CASE iStopStandby OF
0:
	StandbyStopR(CLK:=stopStandby);
	IF StandbyStopR.Q THEN
		iStopStandby := 5;
	END_IF
5:
	IF FSMode THEN
		FSStopStandby(IN:=TRUE,PT:=FSTime);
		IF FSStopStandby.Q THEN
			iStopStandby := 10;
			FSStopStandby(IN:=FALSE,PT:=FSTime);
		END_IF
	ELSE
		iStopStandby:=10;
	END_IF
10:
	standbyCommand := FALSE;
	stopStandbyTimer(IN:=TRUE, PT:=timeout);
		IF stopStandbyTimer.Q THEN
			stopStandbyTimer(IN:=FALSE);
			IF NOT standbyClose THEN
				IF standbyStart THEN
					criticalStandbyStopFailed := TRUE;
				END_IF
					warningStandbyNotClose := TRUE;
			END_IF
			iStopStandby := 0;
		END_IF
END_CASE


(*-------------------------------------------------------------------------------------------------------------------------------------------*)

CASE iStopThird OF
0:
	ThirdStopR(CLK:=stopThird);
	IF ThirdStopR.Q THEN
		iStopThird := 10;
	END_IF
10:
	thirdCommand := FALSE;
	stopThirdTimer(IN:=TRUE, PT:=timeout);
		IF stopThirdTimer.Q THEN
			stopThirdTimer(IN:=FALSE);
			IF NOT thirdClose THEN
				IF thirdStart THEN
					criticalThirdStopFailed := TRUE;
				END_IF
				warningThirdNotClose := TRUE;
			END_IF
			iStopThird := 0;
		END_IF
END_CASE


(*-------------------------------------------------------------------------------------------------------------------------------------------*)

SOnceDuty(CLK:=(iStopDuty = 10));
IF SOnceDuty.Q THEN
		A1^:=FALSE;
		A2^:=FALSE;
		A3^:=FALSE;
END_IF


SOnceStandby(CLK:=(iStopStandby = 10));
IF SOnceStandby.Q THEN
		B1^:=FALSE;
		B2^:=FALSE;
		B3^:=FALSE;
END_IF

IF thirdDevice THEN
SOnceThird(CLK:=(iStopThird = 10));
IF SOnceThird.Q THEN
		C1^:=FALSE;
		C2^:=FALSE;
		C3^:=FALSE;
END_IF
END_IF


(*-------------------------------------------------------------------------------------------------------------------------------------------*)

(*
IF FSMode THEN

FSBothStop(IN:=NOT dutyCommand AND NOT standbyCommand,PT:=FSBothTime);
SOnceFS(CLK:=FSBothStop.Q);
IF SOnceFS.Q THEN
	FSBothStop(IN:=FALSE,PT:=FSBothTime);
	Q1^ := TRUE;
	Q2^ := TRUE;
	Q3^:=TRUE;
END_IF

END_IF
*)
END_ACTION
ACTION test:
dutyStart := dutyCommand;
standbyStart := standbyCommand;
thirdStart:=thirdCommand;
END_ACTION

(* POU module/INLET_SCREENING_OPERATION_2_old, CFC *)
PROGRAM INLET_SCREENING_OPERATION_2_old
VAR
	bTest: BOOL;
	bTestReault: BOOL;

	LSH105B : inBlock;
	LSHH105B: inBlock;
	bPenstockDual: BOOL;
	Timer1: TON;
	bWarningStreamLineOverflow: BOOL;
	bFineScreen: BOOL;
	F101B: fb_equipment_with_linking;
	XV101B1 : fb_equipment_with_linking;
	StopTimer: TON;
	bScrewConveyor: BOOL;
	bScreenCompactor: BOOL;
	bWaterSprayScreenDuty: BOOL;
	bWaterSprayScreenStandby: BOOL;
	bPenstockDuty: BOOL;
	bPenstockStandby: BOOL;
	XV101B2: fb_equipment_with_linking;
	timerCompactor: TON;
	bFineScreenDual: BOOL;
	PS101B: fb_equipment_with_linking;
	bContinuousWaterSpray: BOOL;
	C102B: fb_equipment_with_linking;
	C101B: fb_equipment_with_linking;
	XV102B: fb_equipment_with_linking;
END_VAR
VAR (* helpers for the ST form of the networks *)
	_en57 : BOOL;
	_t57 : BOOL;
	_en85 : BOOL;
	_t85 : BOOL;
END_VAR
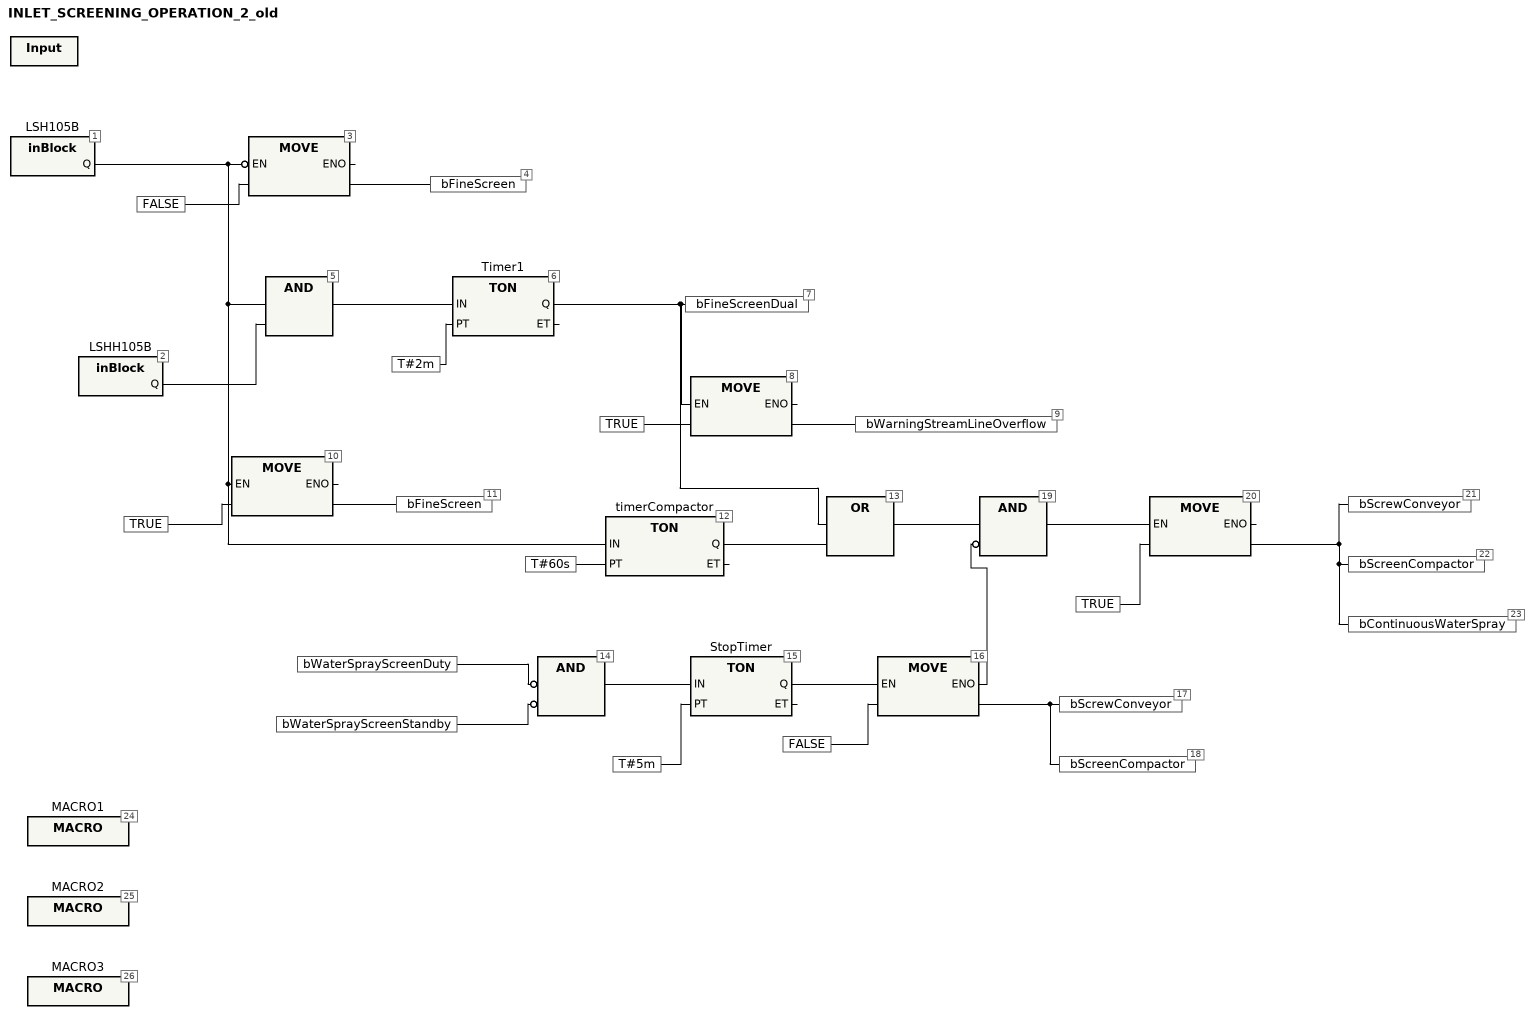
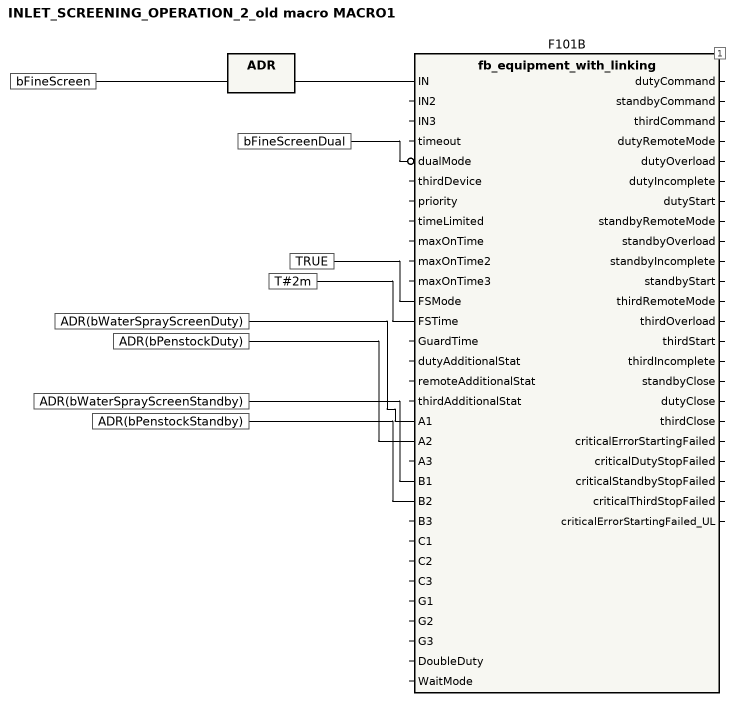
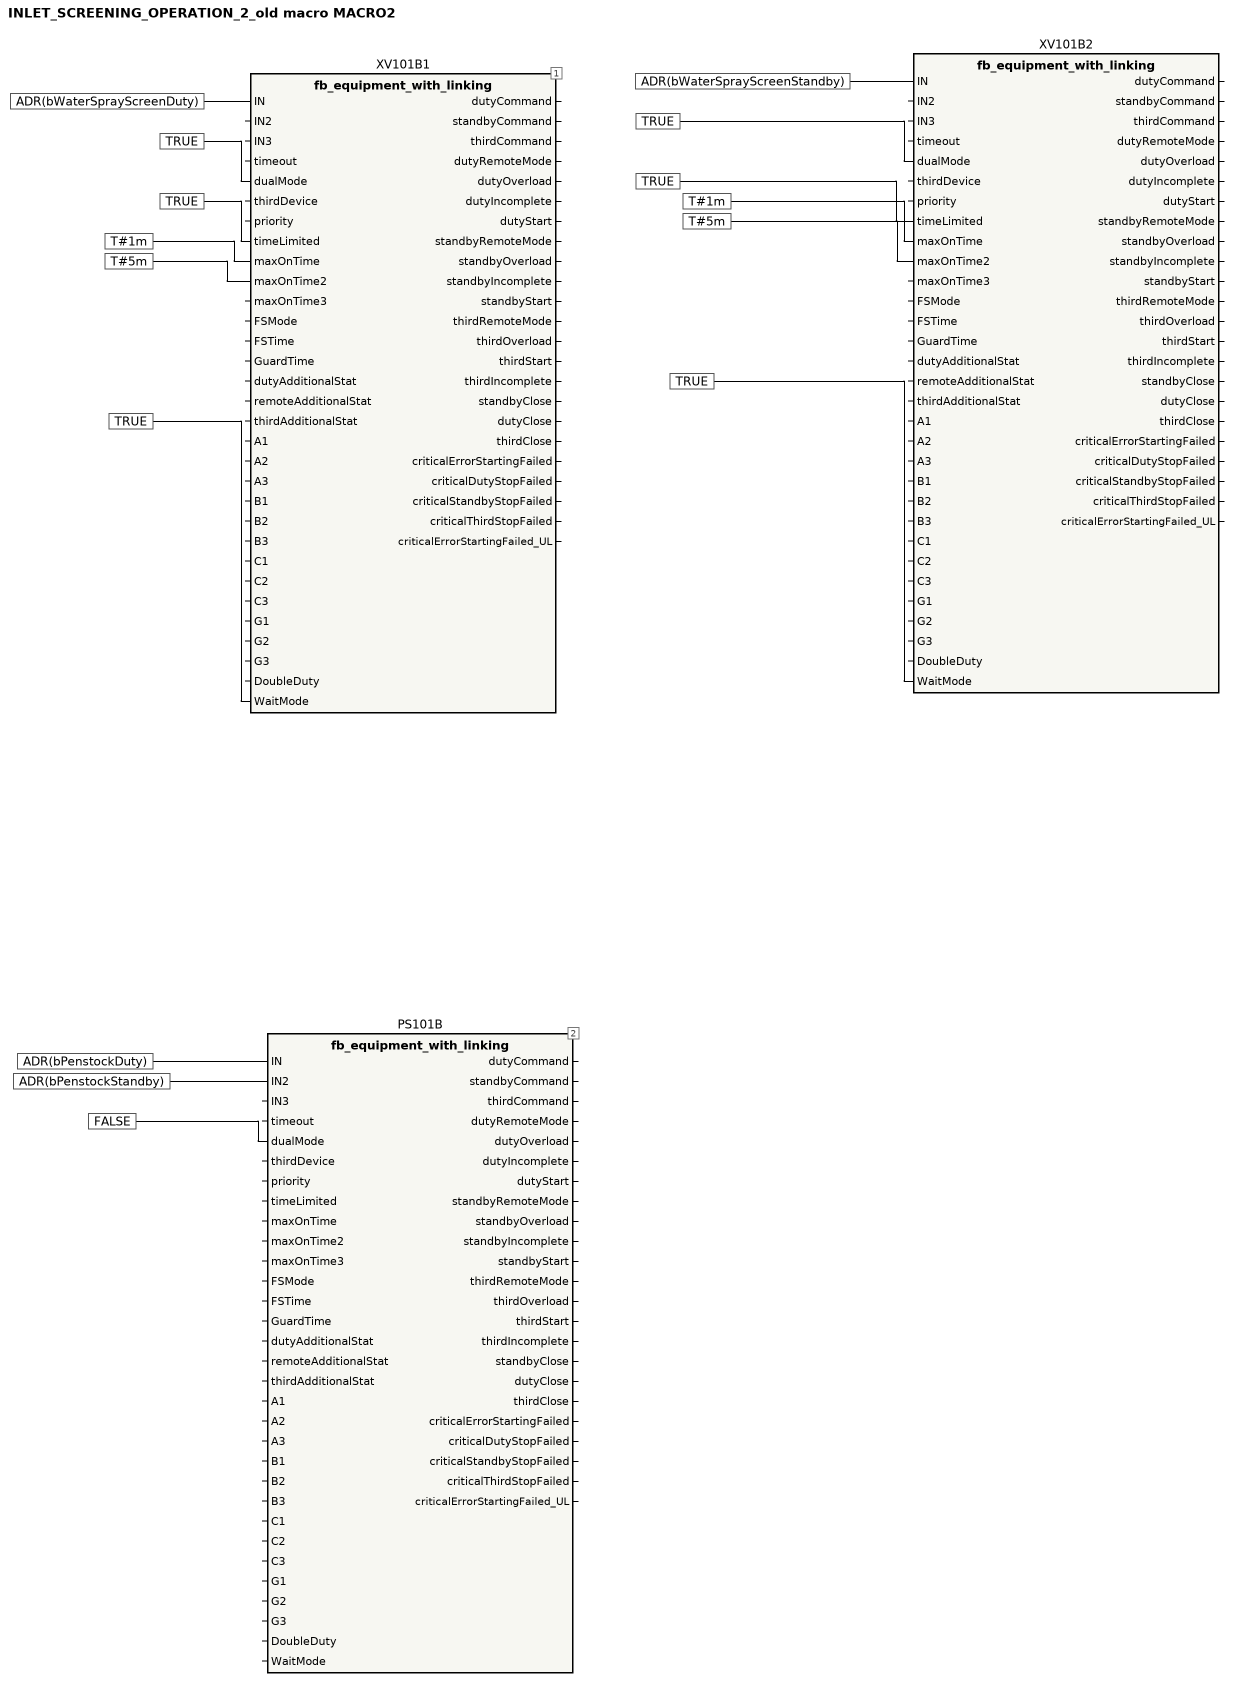
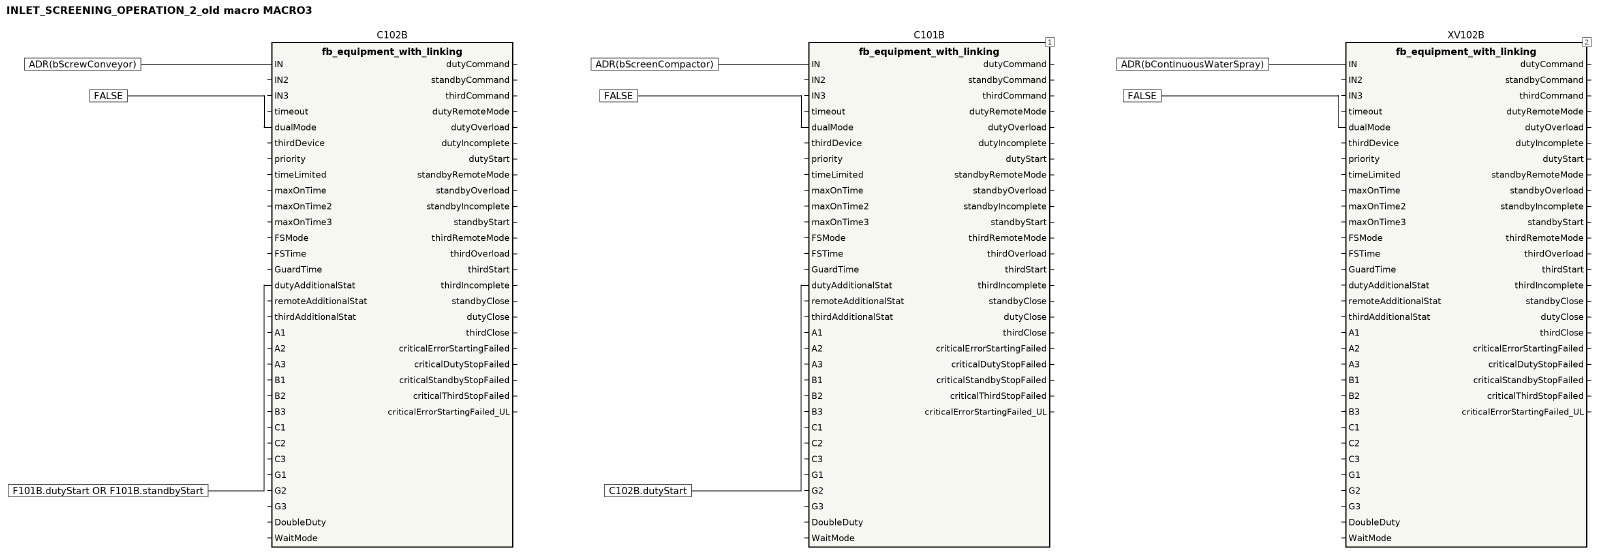
_CFC_ (* Continuous Function Chart, elements in execution order *)
#0 Input()
#1 LSH105B:inBlock()
#2 LSHH105B:inBlock()
#3 MOVE(EN: NOT #1.Q, FALSE)
#4 bFineScreen <= #3
#5 AND(#1.Q, #2.Q)
#6 Timer1:TON(IN: #5, PT: T#2m)
#7 bFineScreenDual <= #6.Q
#8 MOVE(EN: #6.Q, TRUE)
#9 bWarningStreamLineOverflow <= #8
#10 MOVE(EN: #1.Q, TRUE)
#11 bFineScreen <= #10
#12 timerCompactor:TON(IN: #1.Q, PT: T#60s)
#13 OR(#6.Q, #12.Q)
#14 AND(NOT bWaterSprayScreenDuty, NOT bWaterSprayScreenStandby)
#15 StopTimer:TON(IN: #14, PT: T#5m)
#16 MOVE(EN: #15.Q, FALSE)
#17 bScrewConveyor <= #16
#18 bScreenCompactor <= #16
#19 AND(#13, NOT #16.ENO)
#20 MOVE(EN: #19, TRUE)
#21 bScrewConveyor <= #20
#22 bScreenCompactor <= #20
#23 bContinuousWaterSpray <= #20
#24 MACRO MACRO1()
	#25 ADR(bFineScreen)
	#26 F101B:fb_equipment_with_linking(IN: #25, IN2: -, IN3: -, timeout: -, dualMode: NOT bFineScreenDual, thirdDevice: -, priority: -, timeLimited: -, maxOnTime: -, maxOnTime2: -, maxOnTime3: -, FSMode: TRUE, FSTime: T#2m, GuardTime: -, dutyAdditionalStat: -, remoteAdditionalStat: -, thirdAdditionalStat: -, A1: ADR(bWaterSprayScreenDuty), A2: ADR(bPenstockDuty), A3: -, B1: ADR(bWaterSprayScreenStandby), B2: ADR(bPenstockStandby), B3: -, C1: -, C2: -, C3: -, G1: -, G2: -, G3: -, DoubleDuty: -, WaitMode: -)
END_MACRO
#27 MACRO MACRO2()
	#28 XV101B2:fb_equipment_with_linking(IN: ADR(bWaterSprayScreenStandby), IN2: -, IN3: -, timeout: -, dualMode: TRUE, thirdDevice: -, priority: -, timeLimited: TRUE, maxOnTime: T#1m, maxOnTime2: T#5m, maxOnTime3: -, FSMode: -, FSTime: -, GuardTime: -, dutyAdditionalStat: -, remoteAdditionalStat: -, thirdAdditionalStat: -, A1: -, A2: -, A3: -, B1: -, B2: -, B3: -, C1: -, C2: -, C3: -, G1: -, G2: -, G3: -, DoubleDuty: -, WaitMode: TRUE)
	#29 XV101B1:fb_equipment_with_linking(IN: ADR(bWaterSprayScreenDuty), IN2: -, IN3: -, timeout: -, dualMode: TRUE, thirdDevice: -, priority: -, timeLimited: TRUE, maxOnTime: T#1m, maxOnTime2: T#5m, maxOnTime3: -, FSMode: -, FSTime: -, GuardTime: -, dutyAdditionalStat: -, remoteAdditionalStat: -, thirdAdditionalStat: -, A1: -, A2: -, A3: -, B1: -, B2: -, B3: -, C1: -, C2: -, C3: -, G1: -, G2: -, G3: -, DoubleDuty: -, WaitMode: TRUE)
	#30 PS101B:fb_equipment_with_linking(IN: ADR(bPenstockDuty), IN2: ADR(bPenstockStandby), IN3: -, timeout: -, dualMode: FALSE, thirdDevice: -, priority: -, timeLimited: -, maxOnTime: -, maxOnTime2: -, maxOnTime3: -, FSMode: -, FSTime: -, GuardTime: -, dutyAdditionalStat: -, remoteAdditionalStat: -, thirdAdditionalStat: -, A1: -, A2: -, A3: -, B1: -, B2: -, B3: -, C1: -, C2: -, C3: -, G1: -, G2: -, G3: -, DoubleDuty: -, WaitMode: -)
END_MACRO
#31 MACRO MACRO3()
	#32 C102B:fb_equipment_with_linking(IN: ADR(bScrewConveyor), IN2: -, IN3: -, timeout: -, dualMode: FALSE, thirdDevice: -, priority: -, timeLimited: -, maxOnTime: -, maxOnTime2: -, maxOnTime3: -, FSMode: -, FSTime: -, GuardTime: -, dutyAdditionalStat: F101B.dutyStart OR F101B.standbyStart, remoteAdditionalStat: -, thirdAdditionalStat: -, A1: -, A2: -, A3: -, B1: -, B2: -, B3: -, C1: -, C2: -, C3: -, G1: -, G2: -, G3: -, DoubleDuty: -, WaitMode: -)
	#33 C101B:fb_equipment_with_linking(IN: ADR(bScreenCompactor), IN2: -, IN3: -, timeout: -, dualMode: FALSE, thirdDevice: -, priority: -, timeLimited: -, maxOnTime: -, maxOnTime2: -, maxOnTime3: -, FSMode: -, FSTime: -, GuardTime: -, dutyAdditionalStat: C102B.dutyStart, remoteAdditionalStat: -, thirdAdditionalStat: -, A1: -, A2: -, A3: -, B1: -, B2: -, B3: -, C1: -, C2: -, C3: -, G1: -, G2: -, G3: -, DoubleDuty: -, WaitMode: -)
	#34 XV102B:fb_equipment_with_linking(IN: ADR(bContinuousWaterSpray), IN2: -, IN3: -, timeout: -, dualMode: FALSE, thirdDevice: -, priority: -, timeLimited: -, maxOnTime: -, maxOnTime2: -, maxOnTime3: -, FSMode: -, FSTime: -, GuardTime: -, dutyAdditionalStat: -, remoteAdditionalStat: -, thirdAdditionalStat: -, A1: -, A2: -, A3: -, B1: -, B2: -, B3: -, C1: -, C2: -, C3: -, G1: -, G2: -, G3: -, DoubleDuty: -, WaitMode: -)
END_MACRO
_END_CFC_
(* the same logic as Structured Text *)
Input();
LSH105B();
LSHH105B();
IF NOT LSH105B.Q THEN bFineScreen := FALSE; END_IF;
Timer1(IN := LSH105B.Q AND LSHH105B.Q, PT := T#2m);
bFineScreenDual := Timer1.Q;
IF Timer1.Q THEN bWarningStreamLineOverflow := TRUE; END_IF;
IF LSH105B.Q THEN bFineScreen := TRUE; END_IF;
timerCompactor(IN := LSH105B.Q, PT := T#60s);
StopTimer(IN := NOT bWaterSprayScreenDuty AND NOT bWaterSprayScreenStandby, PT := T#5m);
_en57 := StopTimer.Q;
IF _en57 THEN _t57 := FALSE; END_IF;
IF _en57 THEN bScrewConveyor := _t57; END_IF;
IF _en57 THEN bScreenCompactor := _t57; END_IF;
_en85 := (Timer1.Q OR timerCompactor.Q) AND NOT _en57;
IF _en85 THEN _t85 := TRUE; END_IF;
IF _en85 THEN bScrewConveyor := _t85; END_IF;
IF _en85 THEN bScreenCompactor := _t85; END_IF;
IF _en85 THEN bContinuousWaterSpray := _t85; END_IF;
(* macro MACRO1 *)
F101B(IN := ADR(bFineScreen), dualMode := NOT bFineScreenDual, FSMode := TRUE, FSTime := T#2m, A1 := ADR(bWaterSprayScreenDuty), A2 := ADR(bPenstockDuty), B1 := ADR(bWaterSprayScreenStandby), B2 := ADR(bPenstockStandby));
(* macro MACRO2 *)
XV101B2(IN := ADR(bWaterSprayScreenStandby), dualMode := TRUE, timeLimited := TRUE, maxOnTime := T#1m, maxOnTime2 := T#5m, WaitMode := TRUE);
XV101B1(IN := ADR(bWaterSprayScreenDuty), dualMode := TRUE, timeLimited := TRUE, maxOnTime := T#1m, maxOnTime2 := T#5m, WaitMode := TRUE);
PS101B(IN := ADR(bPenstockDuty), IN2 := ADR(bPenstockStandby), dualMode := FALSE);
(* macro MACRO3 *)
C102B(IN := ADR(bScrewConveyor), dualMode := FALSE, dutyAdditionalStat := F101B.dutyStart OR F101B.standbyStart);
C101B(IN := ADR(bScreenCompactor), dualMode := FALSE, dutyAdditionalStat := C102B.dutyStart);
XV102B(IN := ADR(bContinuousWaterSpray), dualMode := FALSE);
END_PROGRAM
ACTION Input:
LSH105B( );
LSHH105B( );
END_ACTION

(* POU module/SLUDGE_THICKENING_SELFIE, CFC *)
PROGRAM SLUDGE_THICKENING_SELFIE
VAR
	SludgeTankLevel_LSL501A: inBlock;
	SludgeTankLevel_LSH501A: inBlock;
	SludePitSensor_LSH600: inBlock;
	PressureSwitch_PSL505A: BOOL;
	SludgeFeedPump_P501A: BOOL;
	DrumThickener_D503A: BOOL;
	BackWashWaterPump_P505A: BOOL;
	Blower_P505A: BOOL;
	PolymerTimerA: TON;
	PolimerTank_LSLPU501: inBlock;
	PolimerTank_LSHPU501: inBlock;
	PolimerValveOpen_XVPU501A: BOOL;
	PolimerValveClose_XVPU501A: BOOL;
	DiagramValvaOpen_XVPU502A: BOOL;

	SludgeTankLevel_LSL501B: inBlock;
	SludgeTankLevel_LSH501B: inBlock;
	PressureSwitch_PSL505B: BOOL;
	SludgeFeedPump_P501B: BOOL;
	DrumThickener_D503B: BOOL;
	BackWashWaterPump_P505B: BOOL;
	Blower_P505B: BOOL;
	PolymerTimerB: TON;
	PolimerValveOpen_XVPU501B: BOOL;
	PolimerValveClose_XVPU501B: BOOL;
	DiagramValvaOpen_XVPU502B: BOOL;


	bWarning_PolimerLow: BOOL;
	DiagramValvaOpen_XVPU502 AT %Q*: BOOL;
	FilterateSumpLevel_LSL620: inBlock;
	FilterateSumpLevel_LSH620: inBlock;
	FilteratePump_P602A: BOOL;
	FilteratePump_P602B: BOOL;
END_VAR
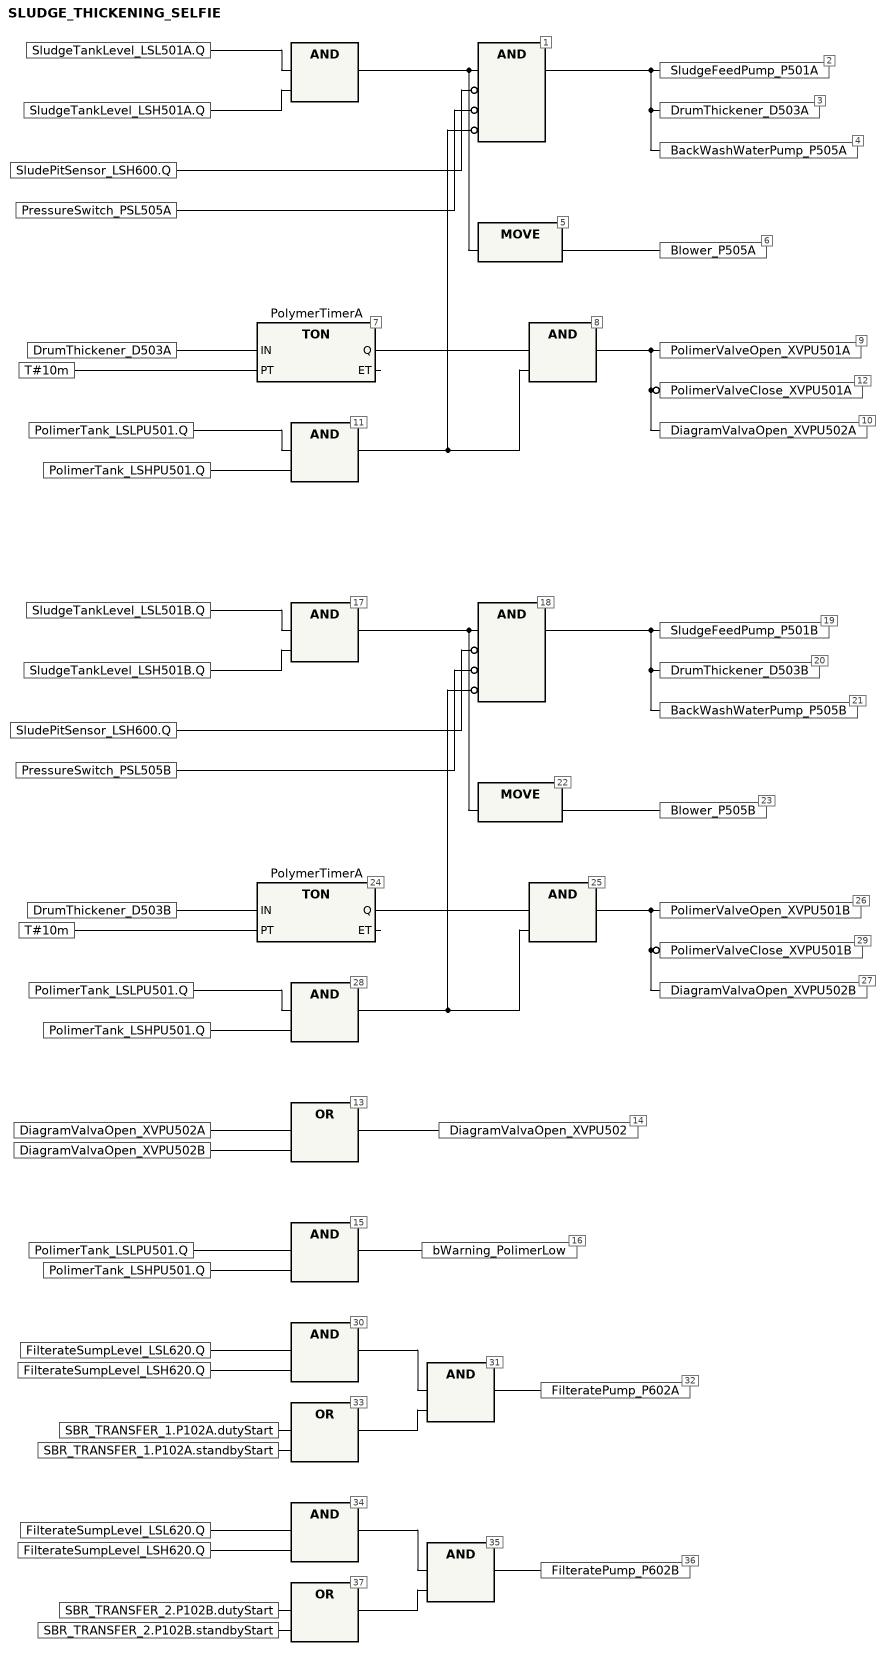
_CFC_ (* Continuous Function Chart, elements in execution order *)
#0 AND(SludgeTankLevel_LSL501A.Q, SludgeTankLevel_LSH501A.Q)
#1 AND(#0, NOT SludePitSensor_LSH600.Q, NOT PressureSwitch_PSL505A, NOT #11)
#2 SludgeFeedPump_P501A <= #1
#3 DrumThickener_D503A <= #1
#4 BackWashWaterPump_P505A <= #1
#5 MOVE(#0)
#6 Blower_P505A <= #5
#7 PolymerTimerA:TON(IN: DrumThickener_D503A, PT: T#10m)
#8 AND(#7.Q, #11)
#9 PolimerValveOpen_XVPU501A <= #8
#10 DiagramValvaOpen_XVPU502A <= #8
#11 AND(PolimerTank_LSLPU501.Q, PolimerTank_LSHPU501.Q)
#12 PolimerValveClose_XVPU501A <= NOT #8
#13 OR(DiagramValvaOpen_XVPU502A, DiagramValvaOpen_XVPU502B)
#14 DiagramValvaOpen_XVPU502 <= #13
#15 AND(PolimerTank_LSLPU501.Q, PolimerTank_LSHPU501.Q)
#16 bWarning_PolimerLow <= #15
#17 AND(SludgeTankLevel_LSL501B.Q, SludgeTankLevel_LSH501B.Q)
#18 AND(#17, NOT SludePitSensor_LSH600.Q, NOT PressureSwitch_PSL505B, NOT #28)
#19 SludgeFeedPump_P501B <= #18
#20 DrumThickener_D503B <= #18
#21 BackWashWaterPump_P505B <= #18
#22 MOVE(#17)
#23 Blower_P505B <= #22
#24 PolymerTimerA:TON(IN: DrumThickener_D503B, PT: T#10m)
#25 AND(#24.Q, #28)
#26 PolimerValveOpen_XVPU501B <= #25
#27 DiagramValvaOpen_XVPU502B <= #25
#28 AND(PolimerTank_LSLPU501.Q, PolimerTank_LSHPU501.Q)
#29 PolimerValveClose_XVPU501B <= NOT #25
#30 AND(FilterateSumpLevel_LSL620.Q, FilterateSumpLevel_LSH620.Q)
#31 AND(#30, #33)
#32 FilteratePump_P602A <= #31
#33 OR(SBR_TRANSFER_1.P102A.dutyStart, SBR_TRANSFER_1.P102A.standbyStart)
#34 AND(FilterateSumpLevel_LSL620.Q, FilterateSumpLevel_LSH620.Q)
#35 AND(#34, #37)
#36 FilteratePump_P602B <= #35
#37 OR(SBR_TRANSFER_2.P102B.dutyStart, SBR_TRANSFER_2.P102B.standbyStart)
_END_CFC_
END_PROGRAM

(* POU module/STREAM_INLET_MIXER_2_OLD, CFC *)
PROGRAM STREAM_INLET_MIXER_2_OLD
VAR
	LSL101B : inBlock;
	LSS101B : inBlock;
	LSH101B : inBlock;
	LSD101B : inBlock;

	LSL100B : inBlock;
	LSHL100B:inBlock;

	bEQPump: BOOL;
	bCriticalEQFloatHi: BOOL;
	bWarningFloatSensorLow: BOOL;
	bCriticalFloatSensorDry: BOOL;
	bEQMixer: BOOL;
	P101B: fb_equipment_with_linking;
	M101B: fb_equipment_with_linking;
END_VAR
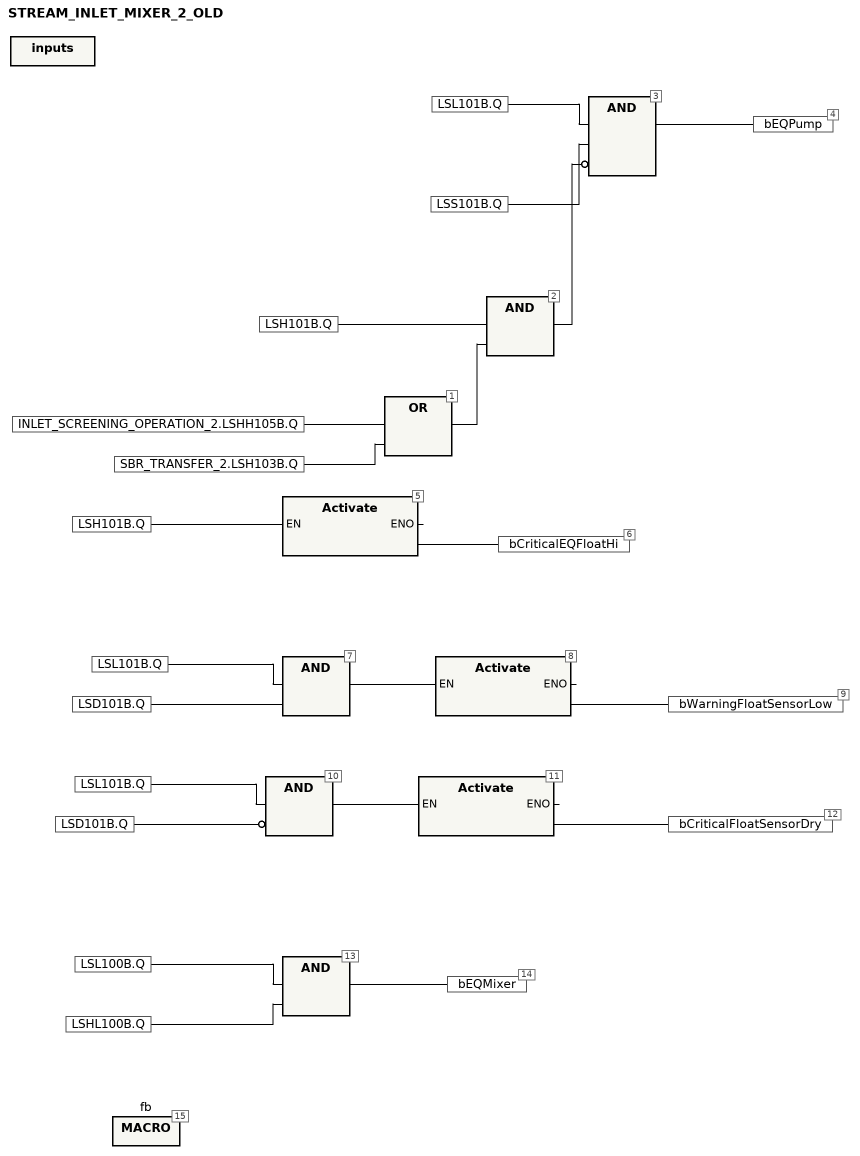
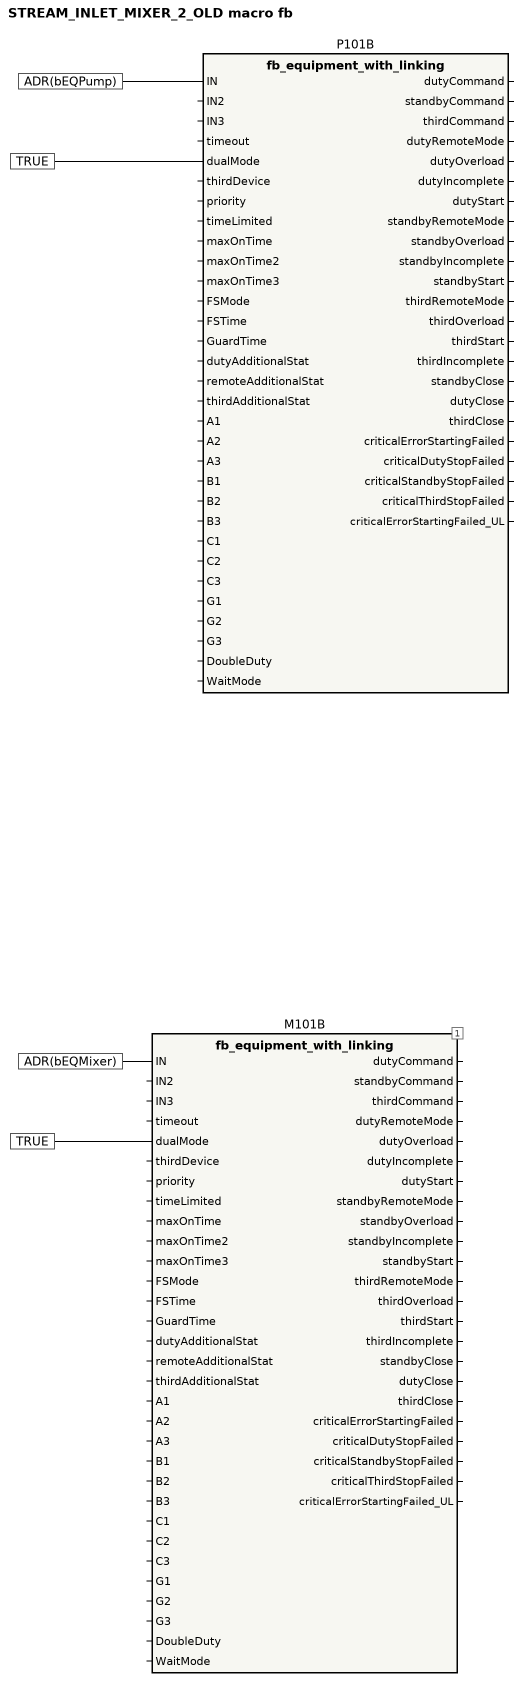
_CFC_ (* Continuous Function Chart, elements in execution order *)
#0 inputs()
#1 OR(INLET_SCREENING_OPERATION_2.LSHH105B.Q, SBR_TRANSFER_2.LSH103B.Q)
#2 AND(LSH101B.Q, #1)
#3 AND(LSL101B.Q, LSS101B.Q, NOT #2)
#4 bEQPump <= #3
#5 Activate(EN: LSH101B.Q)
#6 bCriticalEQFloatHi <= #5
#7 AND(LSL101B.Q, LSD101B.Q)
#8 Activate(EN: #7)
#9 bWarningFloatSensorLow <= #8
#10 AND(LSL101B.Q, NOT LSD101B.Q)
#11 Activate(EN: #10)
#12 bCriticalFloatSensorDry <= #11
#13 AND(LSL100B.Q, LSHL100B.Q)
#14 bEQMixer <= #13
#15 MACRO fb()
	#16 P101B:fb_equipment_with_linking(IN: ADR(bEQPump), IN2: -, IN3: -, timeout: -, dualMode: TRUE, thirdDevice: -, priority: -, timeLimited: -, maxOnTime: -, maxOnTime2: -, maxOnTime3: -, FSMode: -, FSTime: -, GuardTime: -, dutyAdditionalStat: -, remoteAdditionalStat: -, thirdAdditionalStat: -, A1: -, A2: -, A3: -, B1: -, B2: -, B3: -, C1: -, C2: -, C3: -, G1: -, G2: -, G3: -, DoubleDuty: -, WaitMode: -)
	#17 M101B:fb_equipment_with_linking(IN: ADR(bEQMixer), IN2: -, IN3: -, timeout: -, dualMode: TRUE, thirdDevice: -, priority: -, timeLimited: -, maxOnTime: -, maxOnTime2: -, maxOnTime3: -, FSMode: -, FSTime: -, GuardTime: -, dutyAdditionalStat: -, remoteAdditionalStat: -, thirdAdditionalStat: -, A1: -, A2: -, A3: -, B1: -, B2: -, B3: -, C1: -, C2: -, C3: -, G1: -, G2: -, G3: -, DoubleDuty: -, WaitMode: -)
END_MACRO
_END_CFC_
(* the same logic as Structured Text *)
inputs();
bEQPump := LSL101B.Q AND LSS101B.Q AND NOT (LSH101B.Q AND (INLET_SCREENING_OPERATION_2.LSHH105B.Q OR SBR_TRANSFER_2.LSH103B.Q));
IF LSH101B.Q THEN bCriticalEQFloatHi := Activate(); END_IF;
IF LSL101B.Q AND LSD101B.Q THEN bWarningFloatSensorLow := Activate(); END_IF;
IF LSL101B.Q AND NOT LSD101B.Q THEN bCriticalFloatSensorDry := Activate(); END_IF;
bEQMixer := LSL100B.Q AND LSHL100B.Q;
(* macro fb *)
P101B(IN := ADR(bEQPump), dualMode := TRUE);
M101B(IN := ADR(bEQMixer), dualMode := TRUE);
END_PROGRAM
ACTION inputs:
	LSL101B();
	LSS101B();
	LSH101B();
	LSD101B();

	LSL100B();
	LSHL100B();
END_ACTION

(* POU module/TANK_FOR_STREAM_1, ST *)
PROGRAM TANK_FOR_STREAM_1
VAR

(* ---------------------------------------- INLET EQ PUMP OPERATION------------------------------------*)
	LSD101A : inBlock;
	LSL101A : inBlock;
	LSS101A : inBlock;
	LSH101A : inBlock;
	LSHH105A : inBlock;
	LSH103A : inBlock;

	P101A: BOOL;

	warning_EQFloatSensorDry: BOOL;
	critical_EQFloatSensorDry: BOOL;
	critical_EQFloatSensorHi: BOOL;

	fbP101A : fb_equipment;
	P101A1RemoteMode AT%I*: BOOL;
	P101A1Overload AT%I*: BOOL;
	P101A1Incomplete AT%I*: BOOL;
	P101A1Started AT%I*: BOOL;
	P101A2RemoteMode AT%I*: BOOL;
	P101A2Overload AT%I*: BOOL;
	P101A2Incomplete AT%I*: BOOL;
	P101A2Started AT%I*: BOOL;
	warning_P101A1Overload: BOOL;
	warning_P101A1Failed: BOOL;
	warning_P101A2Overload: BOOL;
	warning_P101A2Failed: BOOL;
	critical_P101AStartingFailed: BOOL;
	critical_P101A1StopFailed: BOOL;
	critical_P101A2StopFailed: BOOL;

	P101A1Command AT%Q*: BOOL;
	P101A2Command AT%Q*: BOOL;


(*--------------------------------------------------MIXER Operation-------------------------------------------------*)
	fbM101A : fb_equipment;
	M101A : BOOL;

	M101A1RemoteMode AT%I*: BOOL;
	M101A1Overload AT%I*: BOOL;
	M101A1Incomplete AT%I*: BOOL;
	M101A1Started AT%I*: BOOL;
	M101A2RemoteMode AT%I*: BOOL;
	M101A2Overload AT%I*: BOOL;
	M101A2Incomplete AT%I*: BOOL;
	M101A2Started AT%I*: BOOL;
	warning_M101A1Overload: BOOL;
	warning_M101A1Failed: BOOL;
	warning_M101A2Overload: BOOL;
	warning_M101A2Failed: BOOL;
	critical_M101AStartingFailed: BOOL;
	critical_M101A1StopFailed: BOOL;
	critical_M101A2StopFailed: BOOL;

	M101A1Command AT%Q*: BOOL;
	M101A2Command AT%Q*: BOOL;

	LSL100A : inBlock;
	LSHL100A : inBlock;



END_VAR
LSD101A();
LSL101A();
LSS101A();
LSH101A();
LSHH105A();
LSH103A();

LSL100A();
LSHL100A();



(* ---------------------------------------- INLET EQ PUMP OPERATION------------------------------------*)
fbP101A.IN := ADR(P101A);


IF LSL101A.Q THEN
	IF LSS101A.Q THEN
		P101A:=TRUE;
		IF LSH101A.Q THEN
			critical_EQFloatSensorHi := TRUE;
			IF LSHH105A.Q OR LSH103A.Q THEN
				P101A:=FALSE;
			END_IF
		END_IF
	ELSE
		P101A:=FALSE;
	END_IF
ELSE
	P101A:=FALSE;
	IF LSD101A.Q	THEN
		warning_EQFloatSensorDry :=TRUE;
	ELSE
		critical_EQFloatSensorDry := TRUE;
	END_IF
END_IF

fbP101A(
	dutyRemoteMode:= P101A1RemoteMode,
	dutyOverload:=P101A1Overload ,
	dutyIncomplete:=P101A1Incomplete ,
	dutyStart:=P101A1Started ,
	standbyRemoteMode:=P101A2RemoteMode ,
	standbyOverload:=P101A2Overload ,
	standbyIncomplete:=P101A2Incomplete  ,
	standbyStart:=P101A2Started ,
	timeout:=T#2s ,
	dualMode:= TRUE,
	warningDutyOverload:=ADR(warning_P101A1Overload) ,
	warningDutyFailed:=ADR(warning_P101A1Failed) ,
	warningStandbyOverload:=ADR(warning_P101A2Overload) ,
	warningStandbyFailed:=ADR(warning_P101A2Failed) ,
	criticalErrorStartingFailed:=ADR(critical_P101AStartingFailed) ,
	criticalDutyStopFailed:= ADR(critical_P101A1StopFailed),
	criticalStandbyStopFailed:=ADR(critical_P101A2StopFailed),
	dutyCommand=>P101A1Command ,
	standbyCommand=>P101A2Command);

(*--------------------------------------------------MIXER Operation-------------------------------------------------*)
fbM101A.IN:=ADR(M101A);

IF LSL100A.Q THEN
	IF LSHL100A.Q THEN
		M101A:=TRUE ;
	ELSE
		M101A:=FALSE;
	END_IF
ELSE
	M101A:=FALSE;
END_IF


fbM101A(
	dutyRemoteMode:= M101A1RemoteMode,
	dutyOverload:=M101A1Overload ,
	dutyIncomplete:=M101A1Incomplete ,
	dutyStart:=M101A1Started ,
	standbyRemoteMode:=M101A2RemoteMode ,
	standbyOverload:=M101A2Overload ,
	standbyIncomplete:=M101A2Incomplete  ,
	standbyStart:=M101A2Started ,
	timeout:=T#2s ,
	dualMode:= TRUE,
	warningDutyOverload:=ADR(warning_M101A1Overload) ,
	warningDutyFailed:=ADR(warning_M101A1Failed) ,
	warningStandbyOverload:=ADR(warning_M101A2Overload) ,
	warningStandbyFailed:=ADR(warning_M101A2Failed) ,
	criticalErrorStartingFailed:=ADR(critical_M101AStartingFailed) ,
	criticalDutyStopFailed:= ADR(critical_M101A1StopFailed),
	criticalStandbyStopFailed:=ADR(critical_M101A2StopFailed),
	dutyCommand=>M101A1Command ,
	standbyCommand=>M101A2Command );
END_PROGRAM

(* POU module/fb_equipment, ST *)
FUNCTION_BLOCK fb_equipment
VAR_INPUT
	IN							: POINTER TO BOOL;
	dutyRemoteMode				: BOOL;
	dutyOverload					: BOOL;
	dutyIncomplete				: BOOL;
	dutyStart						: BOOL;

	standbyRemoteMode			: BOOL;
	standbyOverload				: BOOL;
	standbyIncomplete			: BOOL;
	standbyStart					: BOOL;

	thirdRemoteMode				: BOOL;
	thirdOverload					: BOOL;
	thirdStart						: BOOL;
	thirdIncomplete				: BOOL;

	standbyClose					: BOOL;
	dutyClose					: BOOL;
	thirdClose					: BOOL;

	dutyAdditionalStat				: BOOL := TRUE;
	remoteAdditionalStat			: BOOL := TRUE;
	thirdAdditionalStat				: BOOL := TRUE;

	timeout						: TIME:= T#2s;
	dualMode					: BOOL:=TRUE;
	thirdDevice					: BOOL:= FALSE;
	priority						: BOOL := FALSE;
	timeLimited					: BOOL :=FALSE;
	maxOnTime					: TIME := T#10s;
	maxOnTime2					: TIME := T#10s;
	maxOnTime3					: TIME := T#10s;

	FSMode						: BOOL := FALSE;
	FSTime						: TIME := T#2m;
(*
	FSBothTime					: TIME := T#5m;
*)
	GuardTime					: TIME := T#5m;

	A1							: POINTER TO BOOL;
	A2							: POINTER TO BOOL;
	A3							: POINTER TO BOOL;
	B1							: POINTER TO BOOL;
	B2							: POINTER TO BOOL;
	B3							: POINTER TO BOOL;
	C1							: POINTER TO BOOL;
	C2							: POINTER TO BOOL;
	C3							: POINTER TO BOOL;
(*
	Q1							: POINTER TO BOOL;
	Q2							: POINTER TO BOOL;
	Q3							: POINTER TO BOOL;
*)
	G1							: POINTER TO BOOL;
	G2							: POINTER TO BOOL;
	G3							: POINTER TO BOOL;

	warningDutyOverload			: POINTER TO BOOL;
	warningDutyFailed				: POINTER TO BOOL;
	warningDutyNotClose			: POINTER TO BOOL;
	warningDutyClose				: POINTER TO BOOL;
	warningStandbyOverload		: POINTER TO BOOL;
	warningStandbyFailed			: POINTER TO BOOL;
	warningStandbyNotClose		: POINTER TO BOOL;
	warningStandbyClose			: POINTER TO BOOL;
	warningThirdOverload			: POINTER TO BOOL;
	warningThirdFailed			: POINTER TO BOOL;
	warningThirdNotClose			: POINTER TO BOOL;
	warningThirdClose			: POINTER TO BOOL;

	criticalErrorStartingFailed		: POINTER TO BOOL;
	criticalDutyStopFailed			: POINTER TO BOOL;
	criticalStandbyStopFailed		: POINTER TO BOOL;
	criticalThirdStopFailed			: POINTER TO BOOL;

END_VAR
VAR_OUTPUT
	dutyCommand				: BOOL;
	standbyCommand				: BOOL;
	thirdCommand				: BOOL;
END_VAR
VAR
	duty							: INT;
	iStopDuty					: INT;
	state						: INT;
	third							: INT;
	iStopThird					: INT;
	iStopStandby					: INT;
	standby						: INT;
	startDuty						: BOOL;
	startStandby					: BOOL;
	stopStandby					: BOOL;
	stopDuty						: BOOL;
	dutyHalt						: BOOL;
	standbyHalt					: BOOL;
	stopThird					: BOOL;
	startThird					: BOOL;
	thirdHalt						: BOOL;

	dutyTimer					: TON;
	standbyTimer					: TON;
	stopStandbyTimer				: TON;
	stopDutyTimer				: TON;
	FSStopDuty					:TON;
	FSStopStandby				: TON;
	FSBothStop					: TON;
	OnTimer						: TON;
	StandbyOnTimer				: TON;
	thirdTimer					: TON;
	stopThirdTimer				: TON;
	GuardTONDuty				: TON;
	GuardTONStandby			: TON;
	GuardTONThird				: TON;

	ROnce5						: R_TRIG;
	ROnce10					: R_TRIG;
	ROnce20					: R_TRIG;
	SOnceDuty					: R_TRIG;
	SOnceStandby				: R_TRIG;
	SOnceFS					: R_TRIG;
	SOnceThird					: R_TRIG;
	DutyStopR					: R_TRIG;
	StandbyStopR				: R_TRIG;
	ThirdStopR					: R_TRIG;

	internalDummy: BOOL;
	dummyIN: BOOL;
END_VAR
VAR_IN_OUT
END_VAR
IF IN = 0 THEN
	IN := ADR(dummyIN);
END_IF

IF A1 = 0 THEN
	A1 := ADR(internalDummy);
END_IF
IF A2 = 0 THEN
	A2 := ADR(internalDummy);
END_IF
IF A3 = 0 THEN
	A3 := ADR(internalDummy);
END_IF

IF B1 = 0 THEN
	B1 := ADR(internalDummy);
END_IF
IF B2 = 0 THEN
	B2 := ADR(internalDummy);
END_IF
IF B3 = 0 THEN
	B3 := ADR(internalDummy);
END_IF

IF C1 = 0 THEN
	C1 := ADR(internalDummy);
END_IF
IF C2 = 0 THEN
	C2 := ADR(internalDummy);
END_IF
IF C3 = 0 THEN
	C3 := ADR(internalDummy);
END_IF

IF G1 = 0 THEN
	G1 := ADR(internalDummy);
END_IF
IF G2 = 0 THEN
	G2 := ADR(internalDummy);
END_IF
IF G3 = 0 THEN
	G3 := ADR(internalDummy);
END_IF



IF warningDutyOverload = 0 THEN
	warningDutyOverload := ADR(internalDummy);
END_IF
IF warningDutyFailed = 0 THEN
	warningDutyFailed := ADR(internalDummy);
END_IF
IF warningDutyNotClose = 0 THEN
	warningDutyNotClose := ADR(internalDummy);
END_IF
IF warningDutyClose = 0 THEN
	warningDutyClose := ADR(internalDummy);
END_IF



IF warningStandbyOverload = 0 THEN
	warningStandbyOverload := ADR(internalDummy);
END_IF
IF warningStandbyFailed = 0 THEN
	warningStandbyFailed := ADR(internalDummy);
END_IF
IF warningStandbyNotClose = 0 THEN
	warningStandbyNotClose := ADR(internalDummy);
END_IF
IF warningStandbyClose = 0 THEN
	warningStandbyClose := ADR(internalDummy);
END_IF


IF warningThirdOverload = 0 THEN
	warningThirdOverload := ADR(internalDummy);
END_IF
IF warningThirdFailed = 0 THEN
	warningThirdFailed := ADR(internalDummy);
END_IF
IF warningThirdNotClose = 0 THEN
	warningThirdNotClose := ADR(internalDummy);
END_IF
IF warningThirdClose = 0 THEN
	warningThirdClose := ADR(internalDummy);
END_IF


IF criticalErrorStartingFailed = 0 THEN
	criticalErrorStartingFailed := ADR(internalDummy);
END_IF
IF criticalDutyStopFailed = 0 THEN
	criticalDutyStopFailed := ADR(internalDummy);
END_IF
IF criticalStandbyStopFailed = 0 THEN
	criticalStandbyStopFailed := ADR(internalDummy);
END_IF
IF criticalThirdStopFailed = 0 THEN
	criticalThirdStopFailed := ADR(internalDummy);
END_IF

(*---------------------------------------------------------------------------------------------------------------------------*)

IF NOT IN^ THEN
	state := 0;
	stopDuty := TRUE;
	stopStandby := TRUE;

	startDuty:=FALSE;
	startStandby := FALSE;
	IF thirdDevice THEN
		stopThird :=TRUE;
		startThird := FALSE;
	END_IF
ELSIF IN^ AND NOT dualMode THEN
	state := 0;
	stopDuty := FALSE;
	stopStandby := FALSE;

	startDuty:=TRUE;
	startStandby := TRUE;
	IF thirdDevice THEN
		stopThird :=FALSE;
		startThird := TRUE;
	END_IF

	A1^:= TRUE;
	A2^:=TRUE;
	A3^ :=TRUE;
	B1^:= TRUE;
	B2^:=TRUE;
	B3^ :=TRUE;
	C1^:= TRUE;
	C2^:=TRUE;
	C3^ :=TRUE;
END_IF

(*-------------------------------------------------------------------------------------------------------------------------------------------*)

CASE state OF
0:
	state := 5;
5:
	IF NOT DutyHalt AND dutyStart THEN
		stopStandby := TRUE;
		stopThird:=TRUE;
	END_IF

	stopDuty := FALSE;
	startDuty := TRUE;
	IF timeLimited THEN
		OnTimer(IN:=TRUE,PT:=maxOnTime);
	ELSE
		OnTimer(IN:=FALSE,PT:=maxOnTime);
	END_IF
	IF dutyHalt  OR onTimer.Q THEN
		OnTimer(IN:=FALSE,PT:=maxOnTime);
		startDuty := FALSE;
		stopDuty := TRUE;
		state := 10;
	END_IF
10:
	IF NOT StandbyHalt AND standbyStart THEN
		stopDuty := TRUE;
		stopThird:=TRUE;
	END_IF

	stopStandby := FALSE;
	startStandby := TRUE;

	IF timeLimited THEN
		OnTimer(IN:=TRUE,PT:=maxOnTime2);
	ELSE
		OnTimer(IN:=FALSE,PT:=maxOnTime2);
	END_IF
	IF standbyHalt OR onTimer.Q THEN
		OnTimer(IN:=FALSE,PT:=maxOnTime2);
		startStandby := FALSE;
		stopStandby := TRUE;
		IF thirdDevice THEN
			IF priority THEN
				IF dutyIncomplete OR dutyOverload THEN
					state:= 20;
				ELSE
					dutyHalt := FALSE;
					standbyHalt := FALSE;
					state:=0;
				END_IF
			ELSE
				state:= 20;
			END_IF
		ELSE
			IF dutyIncomplete OR dutyOverload THEN
				CriticalErrorStartingFailed^ := TRUE;
			END_IF
			state:=0;
			dutyHalt := FALSE;
			standbyHalt := FALSE;
		END_IF
	END_IF
20:
	IF NOT thirdHalt AND thirdStart THEN
		stopStandby := TRUE;
		stopDuty:=TRUE;
	END_IF

	stopThird := FALSE;
	startThird := TRUE;
	IF timeLimited THEN
		OnTimer(IN:=TRUE,PT:=maxOnTime3);
	ELSE
		OnTimer(IN:=FALSE,PT:=maxOnTime3);
	END_IF
	IF thirdHalt OR OnTimer.Q THEN
		OnTimer(IN:=FALSE,PT:=maxOnTime3);
		startThird := FALSE;
		stopThird := TRUE;
		state := 0;
		IF  (dutyIncomplete OR dutyOverload)  AND (standbyIncomplete OR standbyOverload) THEN
				CriticalErrorStartingFailed^ := TRUE;
		END_IF
		dutyHalt := FALSE;
		standbyHalt := FALSE;
		thirdHalt := FALSE;
	END_IF
END_CASE



(*-------------------------------------------------------------------------------------------------------------------------------------------*)

CASE duty OF
0:
	IF startDuty THEN
		duty := 5;
	END_IF
5:
	IF dutyRemoteMode AND dutyAdditionalStat THEN
		duty := 10;
	ELSE
		duty := 900;
	END_IF
10:
	IF dutyOverload THEN
		warningDutyOverload^ := TRUE;
		dutyHalt := TRUE;
		duty := 40;
	ELSE
		duty := 15;
	END_IF

15:
	duty := 20;
	dutyCommand := TRUE;
20:
	dutyTimer(IN:= TRUE, PT := timeout);
	IF dutyTimer.Q THEN
		dutyTimer(IN:=FALSE);
		duty := 30;
	END_IF
30:

		IF dutyIncomplete OR NOT dutyStart THEN
			warningDutyFailed^ := TRUE;
			dutyHalt := TRUE;
			IF  dutyClose THEN
				warningDutyClose^ := TRUE;
			END_IF
		END_IF
		duty := 40;
40:

	duty := 900;
900:
	duty := 0;
END_CASE

(*----------------------------------------------------------------------------------------------------------------------*)

CASE standby OF
0:
	IF startStandby THEN
		standby := 5;
	END_IF
5:
	IF standbyRemoteMode AND remoteAdditionalStat THEN
		standby := 10;
	ELSE
		standby := 900;
	END_IF
10:
	IF standbyOverload THEN
		warningStandbyOverload^ := TRUE;
		standbyHalt := TRUE;
		standby := 40;
	ELSE
		standby := 15;
	END_IF
15:
		standbyCommand := TRUE;
		standby := 20;
20:
	standbyTimer(IN:= TRUE, PT := timeout);
	IF standbyTimer.Q THEN
		standbyTimer(IN:=FALSE);
		standby := 30;
	END_IF
30:

		IF standbyIncomplete OR NOT standbyStart THEN
			warningStandbyFailed^ := TRUE;
			standbyHalt := TRUE;
			IF  standbyClose THEN
				warningStandbyClose^ := TRUE;
			END_IF
		END_IF
		standby := 40;
40:

	standby := 900;

900:
	standby := 0;
END_CASE

(*-------------------------------------------------------------------------------------------------------------------------------------------*)

CASE third OF
0:
	IF startThird THEN
		third := 5;
	END_IF
5:
	IF thirdRemoteMode AND thirdAdditionalStat THEN
		third := 10;
	ELSE
		third := 900;
	END_IF
10:
	IF thirdOverload THEN
		warningThirdOverload^ := TRUE;
		thirdHalt := TRUE;
		third := 40;
	ELSE
		third := 15;
	END_IF
15:
		thirdCommand := TRUE;
		third := 20;
20:
	thirdTimer(IN:= TRUE, PT := timeout);
	IF thirdTimer.Q THEN
		thirdTimer(IN:=FALSE);
		third := 30;
	END_IF
30:

		IF thirdIncomplete OR NOT thirdStart THEN
			warningThirdFailed^ := TRUE;
			thirdHalt := TRUE;
			IF thirdClose THEN
				warningThirdClose^ := TRUE;
			END_IF
		END_IF
		third := 40;
40:

	third := 900;

900:
	third := 0;
END_CASE

(*-------------------------------------------------------------------------------------------------------------------------------------------*)

ROnce5(CLK:=(state=5));
IF ROnce5.Q THEN
		A1^:= TRUE;
		A2^:=TRUE;
		A3^ :=TRUE;
END_IF

ROnce10(CLK:=(state=10));
IF ROnce10.Q THEN
		B1^:= TRUE;
		B2^:= TRUE;
		B3^:= TRUE;
END_IF

IF thirdDevice THEN
ROnce20(CLK:=(state=20));
IF ROnce20.Q THEN
		C1^:= TRUE;
		C2^:= TRUE;
		C3^:= TRUE;
END_IF
END_IF

(*-------------------------------------------------------------------------------------------------------------------------------------------*)
GuardTONDuty(IN:=dutyIncomplete OR dutyOverload OR NOT dutyStart, PT:= GuardTime);
IF GuardTONDuty.Q THEN
	G1^ := TRUE;
END_IF
GuardTONStandby(IN:=standbyIncomplete OR standbyOverload OR NOT standbyStart, PT:= GuardTime);
IF GuardTONStandby.Q THEN
	G2^ := TRUE;
END_IF

IF thirdDevice THEN
GuardTONThird(IN:=thirdIncomplete OR thirdOverload OR NOT thirdStart, PT:= GuardTime);
IF GuardTONThird.q THEN
	G3^ := TRUE;
END_IF
END_IF
(*-------------------------------------------------------------------------------------------------------------------------------------------*)
stopAction;
test();
END_FUNCTION_BLOCK
ACTION stopAction:
CASE iStopDuty OF
0:
(*
	DutyStopR(CLK:=stopDuty);
	IF DutyStopR.Q THEN
		iStopDuty := 5;
	END_IF


5:
*)
	IF FSMode THEN
		FSStopDuty(IN:=TRUE,PT:=FSTime);
		IF FSStopDuty.Q THEN
			iStopDuty := 10;
			FSStopDuty(IN:=FALSE,PT:=FSTime);
		END_IF
	ELSE
		iStopDuty:=10;
	END_IF
10:
	dutyCommand := FALSE;
	stopDutyTimer(IN:=TRUE, PT:=timeout);
		IF stopDutyTimer.Q THEN
			stopDutyTimer(IN:=FALSE);
			IF NOT dutyClose THEN
				IF dutyStart THEN
					criticalDutyStopFailed^ := TRUE;
				END_IF
				warningDutyNotClose^ := TRUE;
			END_IF
			iStopDuty := 0;
		END_IF
END_CASE

(*-------------------------------------------------------------------------------------------------------------------------------------------*)

CASE iStopStandby OF
0:
(*
	StandbyStopR(CLK:=stopStandby);
	IF StandbyStopR.Q THEN
		iStopStandby := 5;
	END_IF
5:
*)
	IF FSMode THEN
		FSStopStandby(IN:=TRUE,PT:=FSTime);
		IF FSStopStandby.Q THEN
			iStopStandby := 10;
			FSStopStandby(IN:=FALSE,PT:=FSTime);
		END_IF
	ELSE
		iStopStandby:=10;
	END_IF
10:
	standbyCommand := FALSE;
	stopStandbyTimer(IN:=TRUE, PT:=timeout);
		IF stopStandbyTimer.Q THEN
			stopStandbyTimer(IN:=FALSE);
			IF NOT standbyClose THEN
				IF standbyStart THEN
					criticalStandbyStopFailed^ := TRUE;
				END_IF
					warningStandbyNotClose^ := TRUE;
			END_IF
			iStopStandby := 0;
		END_IF
END_CASE


(*-------------------------------------------------------------------------------------------------------------------------------------------*)

CASE iStopThird OF
0:
(*
	ThirdStopR(CLK:=stopThird);
	IF ThirdStopR.Q THEN
		iStopThird := 10;
	END_IF
10:
*)
	thirdCommand := FALSE;
	stopThirdTimer(IN:=TRUE, PT:=timeout);
		IF stopThirdTimer.Q THEN
			stopThirdTimer(IN:=FALSE);
			IF NOT thirdClose THEN
				IF thirdStart THEN
					criticalThirdStopFailed^ := TRUE;
				END_IF
				warningThirdNotClose^ := TRUE;
			END_IF
			iStopThird := 0;
		END_IF
END_CASE


(*-------------------------------------------------------------------------------------------------------------------------------------------*)

SOnceDuty(CLK:=(iStopDuty = 10));
IF SOnceDuty.Q THEN
		A1^:=FALSE;
		A2^:=FALSE;
		A3^:=FALSE;
END_IF


SOnceStandby(CLK:=(iStopStandby = 10));
IF SOnceStandby.Q THEN
		B1^:=FALSE;
		B2^:=FALSE;
		B3^:=FALSE;
END_IF

IF thirdDevice THEN
SOnceThird(CLK:=(iStopThird = 10));
IF SOnceThird.Q THEN
		C1^:= FALSE;
		C1^:=FALSE;
		C2^:=FALSE;
		C3^:=FALSE;
END_IF
END_IF


(*-------------------------------------------------------------------------------------------------------------------------------------------*)

(*
IF FSMode THEN

FSBothStop(IN:=NOT dutyCommand AND NOT standbyCommand,PT:=FSBothTime);
SOnceFS(CLK:=FSBothStop.Q);
IF SOnceFS.Q THEN
	FSBothStop(IN:=FALSE,PT:=FSBothTime);
	Q1^ := TRUE;
	Q2^ := TRUE;
	Q3^:=TRUE;
END_IF

END_IF
*)
END_ACTION
ACTION test:
dutyStart := dutyCommand;
standbyStart := standbyCommand;
thirdStart:=thirdCommand;
END_ACTION

(* POU module/TANK_FOR_STREAM_2, ST *)
PROGRAM TANK_FOR_STREAM_2
VAR

(* ---------------------------------------- INLET EQ PUMP OPERATION------------------------------------*)
	LSD101B : inBlock;
	LSL101B : inBlock;
	LSS101B : inBlock;
	LSH101B : inBlock;
	LSHH105B : inBlock;
	LSH103B : inBlock;

	P101B: BOOL;

	warning_EQFloatSensorDry: BOOL;
	critical_EQFloatSensorDry: BOOL;
	critical_EQFloatSensorHi: BOOL;

	fbP101B : fb_equipment;
	P101B1RemoteMode AT%I*: BOOL;
	P101B1Overload AT%I*: BOOL;
	P101B1Incomplete AT%I*: BOOL;
	P101B1Started AT%I*: BOOL;
	P101B2RemoteMode AT%I*: BOOL;
	P101B2Overload AT%I*: BOOL;
	P101B2Incomplete AT%I*: BOOL;
	P101B2Started AT%I*: BOOL;
	warning_P101B1Overload: BOOL;
	warning_P101B1Failed: BOOL;
	warning_P101B2Overload: BOOL;
	warning_P101B2Failed: BOOL;
	critical_P101BStartingFailed: BOOL;
	critical_P101B1StopFailed: BOOL;
	critical_P101B2StopFailed: BOOL;

	P101B1Command AT%Q*: BOOL;
	P101B2Command AT%Q*: BOOL;


(*--------------------------------------------------MIXER Operation-------------------------------------------------*)
	fbM101B : fb_equipment;
	M101B : BOOL;

	M101B1RemoteMode AT%I*: BOOL;
	M101B1Overload AT%I*: BOOL;
	M101B1Incomplete AT%I*: BOOL;
	M101B1Started AT%I*: BOOL;
	M101B2RemoteMode AT%I*: BOOL;
	M101B2Overload AT%I*: BOOL;
	M101B2Incomplete AT%I*: BOOL;
	M101B2Started AT%I*: BOOL;

	warning_M101B1Overload: BOOL;
	warning_M101B1Failed: BOOL;
	warning_M101B2Overload: BOOL;
	warning_M101B2Failed: BOOL;
	critical_M101BStartingFailed: BOOL;
	critical_M101B1StopFailed: BOOL;
	critical_M101B2StopFailed: BOOL;

	M101B1Command AT%Q*: BOOL;
	M101B2Command AT%Q*: BOOL;

	LSL100B : inBlock;
	LSHL100B : inBlock;


END_VAR
LSD101B();
LSL101B();
LSS101B();
LSH101B();
LSHH105B();
LSH103B();

LSL100B();
LSHL100B();



(* ---------------------------------------- INLET EQ PUMP OPERATION------------------------------------*)
fbP101B.IN := ADR(P101B);


IF LSL101B.Q THEN
	IF LSS101B.Q THEN
		P101B:=TRUE;
		IF LSH101B.Q THEN
			critical_EQFloatSensorHi := TRUE;
			IF LSHH105B.Q OR LSH103B.Q THEN
				P101B:=FALSE;
			END_IF
		END_IF
	ELSE
		P101B:=FALSE;
	END_IF
ELSE
	P101B:=FALSE;
	IF LSD101B.Q	THEN
		warning_EQFloatSensorDry :=TRUE;
	ELSE
		critical_EQFloatSensorDry := TRUE;
	END_IF
END_IF

fbP101B(
	dutyRemoteMode:= P101B1RemoteMode,
	dutyOverload:=P101B1Overload ,
	dutyIncomplete:=P101B1Incomplete ,
	dutyStart:=P101B1Started ,
	standbyRemoteMode:=P101B2RemoteMode ,
	standbyOverload:=P101B2Overload ,
	standbyIncomplete:=P101B2Incomplete  ,
	standbyStart:=P101B2Started ,
	timeout:=T#2s ,
	dualMode:= TRUE,
	warningDutyOverload:=ADR(warning_P101B1Overload) ,
	warningDutyFailed:=ADR(warning_P101B1Failed) ,
	warningStandbyOverload:=ADR(warning_P101B2Overload) ,
	warningStandbyFailed:=ADR(warning_P101B2Failed) ,
	criticalErrorStartingFailed:=ADR(critical_P101BStartingFailed) ,
	criticalDutyStopFailed:= ADR(critical_P101B1StopFailed),
	criticalStandbyStopFailed:=ADR(critical_P101B2StopFailed),
	dutyCommand=>P101B1Command ,
	standbyCommand=>P101B2Command );

(*--------------------------------------------------MIXER Operation-------------------------------------------------*)
fbM101B.IN := ADR(M101B);

IF LSL100B.Q THEN
	IF LSHL100B.Q THEN
		M101B:=TRUE;
	ELSE
		M101B:=FALSE;
	END_IF
ELSE
	M101B:=FALSE;
END_IF


fbM101B(
	dutyRemoteMode:= M101B1RemoteMode,
	dutyOverload:=M101B1Overload ,
	dutyIncomplete:=M101B1Incomplete ,
	dutyStart:=M101B1Started ,
	standbyRemoteMode:=M101B2RemoteMode ,
	standbyOverload:=M101B2Overload ,
	standbyIncomplete:=M101B2Incomplete  ,
	standbyStart:=M101B2Started ,
	timeout:=T#2s ,
	dualMode:= TRUE,
	warningDutyOverload:=ADR(warning_M101B1Overload) ,
	warningDutyFailed:=ADR(warning_M101B1Failed) ,
	warningStandbyOverload:=ADR(warning_M101B2Overload) ,
	warningStandbyFailed:=ADR(warning_M101B2Failed) ,
	criticalErrorStartingFailed:=ADR(critical_M101BStartingFailed) ,
	criticalDutyStopFailed:= ADR(critical_M101B1StopFailed),
	criticalStandbyStopFailed:=ADR(critical_M101B2StopFailed),
	dutyCommand=>M101B1Command ,
	standbyCommand=>M101B2Command);





TANK_FOR_STREAM_1.LSD101A.IN;
TANK_FOR_STREAM_1.LSD101A.Q;
END_PROGRAM

(* POU module/blinker, FBD *)
FUNCTION_BLOCK blinker
VAR_INPUT
	IN: BOOL;
	OffTime: TIME := T#5m;
	OnTime: TIME:=T#2m;
END_VAR
VAR_OUTPUT
	Q: BOOL;
END_VAR
VAR
	tmr_off: TON;
	tmr_on: TON;
END_VAR
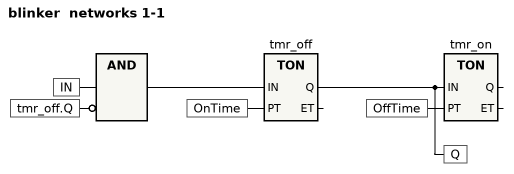
_FBD_ (* Function Block Diagram *)
NETWORK 1
	tmr_on:TON(IN: <tmr_off:TON(IN: AND(IN, NOT tmr_off.Q), PT: OnTime) => Q>, PT: OffTime)
_END_FBD_
END_FUNCTION_BLOCK

(* POU module/ERROR_INTERNAL, CFC *)
FUNCTION_BLOCK ERROR_INTERNAL
VAR_INPUT
	status_error : BOOL;
	trip_error : BOOL;
END_VAR
VAR_OUTPUT
	Q:BOOL;
END_VAR
VAR
	ErrorFilter1: ErrorFilter;
END_VAR
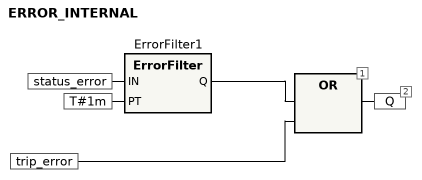
_CFC_ (* Continuous Function Chart, elements in execution order *)
#0 ErrorFilter1:ErrorFilter(IN: status_error, PT: T#1m)
#1 OR(#0.Q, trip_error)
#2 Q <= #1
_END_CFC_
(* the same logic as Structured Text *)
ErrorFilter1(IN := status_error, PT := T#1m);
Q := ErrorFilter1.Q OR trip_error;
END_FUNCTION_BLOCK

(* POU module/fb_equipment_single, ST *)
FUNCTION_BLOCK fb_equipment_single
VAR_INPUT
	IN							: POINTER TO BOOL;

	timeout						: TIME:= T#2s;


	FSMode						: BOOL := FALSE;
	FSTime						: TIME := T#2m;
	GuardTime					: TIME := T#5m;

	A1							: POINTER TO BOOL;
	A2							: POINTER TO BOOL;
	A3							: POINTER TO BOOL;


END_VAR
VAR_OUTPUT

	dutyCommand				AT%Q*: BOOL;

	dutyRemoteMode				AT%I* : BOOL;
	dutyOverload					AT%I* : BOOL;
	dutyIncomplete				AT%I* : BOOL;
	dutyStart						AT%I* : BOOL;

	dutyClose					AT%I* : BOOL;
	dutyAdditionalStat				AT%I* : BOOL := TRUE;


	criticalErrorStartingFailed		: BOOL;
	criticalDutyStopFailed			: BOOL;
	warningDutyOverload			: BOOL;
	warningDutyFailed				: BOOL;
	warningDutyNotClose			: BOOL;
	warningDutyClose				: BOOL;


END_VAR
VAR
	logic :fb_equipment_unlink;
END_VAR
VAR_IN_OUT
END_VAR
logic(
	IN:=IN ,
	IN2:= , 
	IN3:= , 
	timeout:=timeout ,
	dualMode:=FALSE ,
	thirdDevice:=FALSE ,
	priority:=FALSE ,
	timeLimited:=FALSE ,
	maxOnTime:= , 
	maxOnTime2:= ,
	maxOnTime3:= ,
	FSMode:=FALSE ,
	FSTime:= , 
	GuardTime:= , 
	dutyAdditionalStat:=dutyAdditionalStat ,
	remoteAdditionalStat:= , 
	thirdAdditionalStat:= ,
	A1:= A1,
	A2:= A2,
	A3:= A3,
	B1:= , 
	B2:= , 
	B3:= , 
	C1:= , 
	C2:= , 
	C3:= ,
	G1:= , 
	G2:= , 
	G3:= ,
	DoubleDuty:=FALSE ,
	WaitMode:= FALSE,
	dutyCommand:=dutyCommand ,
	standbyCommand:= , 
	thirdCommand:= ,
	dutyRemoteMode:= dutyRemoteMode,
	dutyOverload:= dutyOverload,
	dutyIncomplete:= dutyIncomplete,
	dutyStart:=dutyStart ,
	standbyRemoteMode:= , 
	standbyOverload:= , 
	standbyIncomplete:= , 
	standbyStart:= , 
	thirdRemoteMode:= , 
	thirdOverload:= , 
	thirdStart:= ,
	thirdIncomplete:= , 
	standbyClose:= ,
	dutyClose:= , 
	thirdClose:= ,
	criticalErrorStartingFailed=> criticalErrorStartingFailed,
	criticalDutyStopFailed=>criticalDutyStopFailed ,
	criticalStandbyStopFailed=> , 
	criticalThirdStopFailed=> ,
	criticalErrorStartingFailed_UL=> , 
	warningDutyOverload=>warningDutyOverload ,
	warningDutyFailed=>warningDutyFailed ,
	warningDutyNotClose=>warningDutyNotClose ,
	warningDutyClose=>warningDutyClose ,
	warningStandbyOverload=> , 
	warningStandbyFailed=> , 
	warningStandbyNotClose=> , 
	warningStandbyClose=> , 
	warningThirdOverload=> , 
	warningThirdFailed=> , 
	warningThirdNotClose=> , 
	warningThirdClose=> );
END_FUNCTION_BLOCK

(* POU module/fb_equipment_unlink, ST *)
FUNCTION_BLOCK fb_equipment_unlink
VAR_INPUT
	IN							: POINTER TO BOOL;
	IN2							: POINTER TO BOOL;
	IN3							: POINTER TO BOOL;

	timeout						: TIME:= T#2s;
	dualMode					: BOOL:=TRUE;
	thirdDevice					: BOOL:= FALSE;
	priority						: BOOL := FALSE;
	timeLimited					: BOOL :=FALSE;
	maxOnTime					: TIME := T#10s;
	maxOnTime2					: TIME := T#10s;
	maxOnTime3					: TIME := T#10s;

	FSMode						: BOOL := FALSE;
	FSTime						: TIME := T#2m;
	GuardTime					: TIME := T#5m;




	dutyAdditionalStat			 : BOOL := TRUE;
	remoteAdditionalStat		 : BOOL := TRUE;
	thirdAdditionalStat			 : BOOL := TRUE;

	A1							: POINTER TO BOOL;
	A2							: POINTER TO BOOL;
	A3							: POINTER TO BOOL;
	B1							: POINTER TO BOOL;
	B2							: POINTER TO BOOL;
	B3							: POINTER TO BOOL;
	C1							: POINTER TO BOOL;
	C2							: POINTER TO BOOL;
	C3							: POINTER TO BOOL;
	G1							: POINTER TO BOOL;
	G2							: POINTER TO BOOL;
	G3							: POINTER TO BOOL;

	DoubleDuty: BOOL;
	WaitMode : BOOL;

	dutyCommand				: BOOL;
	standbyCommand				: BOOL;
	thirdCommand				: BOOL;

	dutyRemoteMode				 : BOOL;
	dutyOverload					 : BOOL;
	dutyIncomplete				 : BOOL;
	dutyStart						: BOOL;

	standbyRemoteMode			 : BOOL;
	standbyOverload				 : BOOL;
	standbyIncomplete			: BOOL;
	standbyStart					: BOOL;

	thirdRemoteMode				 : BOOL;
	thirdOverload					 : BOOL;
	thirdStart						 : BOOL;
	thirdIncomplete				 : BOOL;

	standbyClose					 : BOOL;
	dutyClose					 : BOOL;
	thirdClose					 : BOOL;




END_VAR
VAR_OUTPUT


	criticalErrorStartingFailed		: BOOL;
	criticalDutyStopFailed			: BOOL;
	criticalStandbyStopFailed		: BOOL;
	criticalThirdStopFailed			: BOOL;

	criticalErrorStartingFailed_UL	: BOOL;

	warningDutyOverload			: BOOL;
	warningDutyFailed				: BOOL;
	warningDutyNotClose			: BOOL;
	warningDutyClose				: BOOL;
	warningStandbyOverload		: BOOL;
	warningStandbyFailed			: BOOL;
	warningStandbyNotClose		: BOOL;
	warningStandbyClose			: BOOL;
	warningThirdOverload			: BOOL;
	warningThirdFailed			: BOOL;
	warningThirdNotClose			: BOOL;
	warningThirdClose			: BOOL;


END_VAR
VAR


	duty							: INT;
	iStopDuty					: INT;
	state						: INT;
	third							: INT;
	iStopThird					: INT;
	iStopStandby					: INT;
	standby						: INT;
	startDuty						: BOOL;
	startStandby					: BOOL;
	stopStandby					: BOOL;
	stopDuty						: BOOL;
	dutyHalt						: BOOL;
	standbyHalt					: BOOL;
	stopThird					: BOOL;
	startThird					: BOOL;
	thirdHalt						: BOOL;

	dutyTimer					: TON;
	standbyTimer					: TON;
	stopStandbyTimer				: TON;
	stopDutyTimer				: TON;
	FSStopDuty					:TON;
	FSStopStandby				: TON;
	FSBothStop					: TON;
	OnTimer						: TON;
	StandbyOnTimer				: TON;
	thirdTimer					: TON;
	stopThirdTimer				: TON;
	GuardTONDuty				: TON;
	GuardTONStandby			: TON;
	GuardTONThird				: TON;

	ROnce5						: R_TRIG;
	ROnce10					: R_TRIG;
	ROnce20					: R_TRIG;
	SOnceDuty					: R_TRIG;
	SOnceStandby				: R_TRIG;
	SOnceFS					: R_TRIG;
	SOnceThird					: R_TRIG;
	DutyStopR					: R_TRIG;
	StandbyStopR				: R_TRIG;
	ThirdStopR					: R_TRIG;

	internalDummy: BOOL;
	dummyIN: BOOL;
	dummyIN2: BOOL;
	dummyIN3: BOOL;
END_VAR
VAR_IN_OUT
END_VAR
IF WaitMode THEN
	standbyRemoteMode			:=TRUE;

	standbyStart				:=TRUE;

	thirdRemoteMode				:=TRUE;

	thirdIncomplete				:=TRUE;
END_IF

IF IN = 0 THEN
	IN := ADR(dummyIN);
END_IF

IF IN2 = 0 THEN
	IN2 := ADR(dummyIN2);
END_IF

IF IN3 = 0 THEN
	IN3 := ADR(dummyIN3);
END_IF

IF A1 = 0 THEN
	A1 := ADR(internalDummy);
END_IF
IF A2 = 0 THEN
	A2 := ADR(internalDummy);
END_IF
IF A3 = 0 THEN
	A3 := ADR(internalDummy);
END_IF

IF B1 = 0 THEN
	B1 := ADR(internalDummy);
END_IF
IF B2 = 0 THEN
	B2 := ADR(internalDummy);
END_IF
IF B3 = 0 THEN
	B3 := ADR(internalDummy);
END_IF

IF C1 = 0 THEN
	C1 := ADR(internalDummy);
END_IF
IF C2 = 0 THEN
	C2 := ADR(internalDummy);
END_IF
IF C3 = 0 THEN
	C3 := ADR(internalDummy);
END_IF

IF G1 = 0 THEN
	G1 := ADR(internalDummy);
END_IF
IF G2 = 0 THEN
	G2 := ADR(internalDummy);
END_IF
IF G3 = 0 THEN
	G3 := ADR(internalDummy);
END_IF


(*
IF warningDutyOverload = 0 THEN
	warningDutyOverload := ADR(internalDummy);
END_IF
IF warningDutyFailed = 0 THEN
	warningDutyFailed := ADR(internalDummy);
END_IF
IF warningDutyNotClose = 0 THEN
	warningDutyNotClose := ADR(internalDummy);
END_IF
IF warningDutyClose = 0 THEN
	warningDutyClose := ADR(internalDummy);
END_IF



IF warningStandbyOverload = 0 THEN
	warningStandbyOverload := ADR(internalDummy);
END_IF
IF warningStandbyFailed = 0 THEN
	warningStandbyFailed := ADR(internalDummy);
END_IF
IF warningStandbyNotClose = 0 THEN
	warningStandbyNotClose := ADR(internalDummy);
END_IF
IF warningStandbyClose = 0 THEN
	warningStandbyClose := ADR(internalDummy);
END_IF


IF warningThirdOverload = 0 THEN
	warningThirdOverload := ADR(internalDummy);
END_IF
IF warningThirdFailed = 0 THEN
	warningThirdFailed := ADR(internalDummy);
END_IF
IF warningThirdNotClose = 0 THEN
	warningThirdNotClose := ADR(internalDummy);
END_IF
IF warningThirdClose = 0 THEN
	warningThirdClose := ADR(internalDummy);
END_IF


IF criticalErrorStartingFailed = 0 THEN
	criticalErrorStartingFailed := ADR(internalDummy);
END_IF
IF criticalDutyStopFailed = 0 THEN
	criticalDutyStopFailed := ADR(internalDummy);
END_IF
IF criticalStandbyStopFailed = 0 THEN
	criticalStandbyStopFailed := ADR(internalDummy);
END_IF
IF criticalThirdStopFailed = 0 THEN
	criticalThirdStopFailed := ADR(internalDummy);
END_IF
*)
(*---------------------------------------------------------------------------------------------------------------------------*)

IF dualMode THEN

IF NOT IN^ THEN
	state := 0;
	stopDuty := TRUE;
	stopStandby := TRUE;

	startDuty:=FALSE;
	startStandby := FALSE;
	IF thirdDevice THEN
		stopThird :=TRUE;
		startThird := FALSE;
	END_IF
END_IF

ELSE

state := 0;
startDuty := IN^;
stopDuty := NOT IN^;

startStandby := IN2^;
stopStandby := NOT IN2^;

startThird := IN3^;
stopThird := NOT IN3^;

A1^:=  IN^;
A2^:= IN^;
A3^ := IN^;
B1^:=  IN2^;
B2^:= IN2^;
B3^ := IN2^;
C1^:=  IN3^;
C2^:= IN3^;
C3^ := IN3^;

END_IF

(*
IF NOT IN^ THEN
	state := 0;
	stopDuty := TRUE;
	stopStandby := TRUE;

	startDuty:=FALSE;
	startStandby := FALSE;
	IF thirdDevice THEN
		stopThird :=TRUE;
		startThird := FALSE;
	END_IF
ELSIF IN^ AND NOT dualMode THEN
	state := 0;
	stopDuty := FALSE;
	stopStandby := FALSE;

	startDuty:=TRUE;
	startStandby := TRUE;
	IF thirdDevice THEN
		stopThird :=FALSE;
		startThird := TRUE;
	END_IF

	A1^:= TRUE;
	A2^:=TRUE;
	A3^ :=TRUE;
	B1^:= TRUE;
	B2^:=TRUE;
	B3^ :=TRUE;
	C1^:= TRUE;
	C2^:=TRUE;
	C3^ :=TRUE;
END_IF
*)

(*-------------------------------------------------------------------------------------------------------------------------------------------*)

IF NOT DoubleDuty THEN

CASE state OF
0:
	state := 5;
5:
	IF NOT DutyHalt AND dutyStart THEN
		stopStandby := TRUE;
		stopThird:=TRUE;
	END_IF

	stopDuty := FALSE;
	startDuty := TRUE;
	IF timeLimited THEN
		OnTimer(IN:=TRUE,PT:=maxOnTime);
	ELSE
		OnTimer(IN:=FALSE,PT:=maxOnTime);
	END_IF
	IF dutyHalt  OR onTimer.Q THEN
		OnTimer(IN:=FALSE,PT:=maxOnTime);
		startDuty := FALSE;
		stopDuty := TRUE;
		state := 10;
	END_IF
10:
	IF NOT StandbyHalt AND standbyStart THEN
		stopDuty := TRUE;
		stopThird:=TRUE;
	END_IF

	stopStandby := FALSE;
	startStandby := TRUE;

	IF timeLimited THEN
		OnTimer(IN:=TRUE,PT:=maxOnTime2);
	ELSE
		OnTimer(IN:=FALSE,PT:=maxOnTime2);
	END_IF
	IF standbyHalt OR onTimer.Q THEN
		OnTimer(IN:=FALSE,PT:=maxOnTime2);
		startStandby := FALSE;
		stopStandby := TRUE;
		IF thirdDevice THEN
			IF priority THEN
				IF dutyIncomplete OR dutyOverload THEN
					state:= 20;
				ELSE
					dutyHalt := FALSE;
					standbyHalt := FALSE;
					state:=0;
				END_IF
			ELSE
				state:= 20;
			END_IF
		ELSE
			IF dutyIncomplete OR dutyOverload THEN
				CriticalErrorStartingFailed := TRUE;
			END_IF
			state:=0;
			dutyHalt := FALSE;
			standbyHalt := FALSE;
		END_IF
	END_IF
20:
	IF NOT thirdHalt AND thirdStart THEN
		stopStandby := TRUE;
		stopDuty:=TRUE;
	END_IF

	stopThird := FALSE;
	startThird := TRUE;
	IF timeLimited THEN
		OnTimer(IN:=TRUE,PT:=maxOnTime3);
	ELSE
		OnTimer(IN:=FALSE,PT:=maxOnTime3);
	END_IF
	IF thirdHalt OR OnTimer.Q THEN
		OnTimer(IN:=FALSE,PT:=maxOnTime3);
		startThird := FALSE;
		stopThird := TRUE;
		state := 0;
		IF  (dutyIncomplete OR dutyOverload)  AND (standbyIncomplete OR standbyOverload) THEN
				CriticalErrorStartingFailed := TRUE;
		END_IF
		dutyHalt := FALSE;
		standbyHalt := FALSE;
		thirdHalt := FALSE;
	END_IF
END_CASE

ELSE

thirdDevice := TRUE; (*third device must be enable when double duty*)
dualMode := TRUE; (*dual mode also must be true*)

CASE state OF
0:
	state := 5;
5:
	thirdHalt := FALSE;
	stopStandby := TRUE;
	startStandby := FALSE;

	stopDuty := FALSE;
	startDuty := TRUE;

	stopThird := FALSE;
	startThird := TRUE;

	IF dutyHalt  THEN
		state := 10;
	END_IF


	IF thirdHalt  THEN
		state := 20;
	END_IF
10:
	dutyHalt := FALSE;

	stopStandby := FALSE;
	startStandby := TRUE;

	stopDuty := TRUE;
	startDuty := FALSE;

	stopThird := FALSE;
	startThird := TRUE;

	IF standbyHalt THEN
		state:= 0;
	END_IF
20:
	thirdHalt := FALSE;

	stopStandby := FALSE;
	startStandby := TRUE;

	stopDuty := FALSE;
	startDuty := TRUE;

	stopThird := TRUE;
	startThird := FALSE;

	IF standbyHalt THEN
		state:= 0;
	END_IF
END_CASE


IF NOT(state = 0) AND  (dutyIncomplete OR dutyOverload)  AND (standbyIncomplete OR standbyOverload) AND (thirdIncomplete OR thirdOverload)  THEN
	CriticalErrorStartingFailed := TRUE;
	criticalErrorStartingFailed_UL := TRUE;
ELSE
	criticalErrorStartingFailed_UL := FALSE;
END_IF
END_IF

(*-------------------------------------------------------------------------------------------------------------------------------------------*)

CASE duty OF
0:
	IF startDuty THEN
		duty := 5;
	END_IF
5:
	IF dutyRemoteMode AND dutyAdditionalStat THEN
		duty := 10;
	ELSE
		duty := 900;
	END_IF
10:
	IF dutyOverload THEN
		warningDutyOverload := TRUE;
		dutyHalt := TRUE;
		duty := 40;
	ELSE
		duty := 15;
	END_IF

15:
	duty := 20;
	dutyCommand := TRUE;
20:
	dutyTimer(IN:= TRUE, PT := timeout);
	IF dutyTimer.Q THEN
		dutyTimer(IN:=FALSE);
		duty := 30;
	END_IF
30:

		IF dutyIncomplete OR NOT dutyStart THEN
			warningDutyFailed := TRUE;
			dutyHalt := TRUE;
			IF  dutyClose THEN
				warningDutyClose := TRUE;
			END_IF
		END_IF
		duty := 40;
40:

	duty := 900;
900:
	duty := 0;
END_CASE

(*----------------------------------------------------------------------------------------------------------------------*)

CASE standby OF
0:
	IF startStandby THEN
		standby := 5;
	END_IF
5:
	IF standbyRemoteMode AND remoteAdditionalStat THEN
		standby := 10;
	ELSE
		standby := 900;
	END_IF
10:
	IF standbyOverload THEN
		warningStandbyOverload := TRUE;
		standbyHalt := TRUE;
		standby := 40;
	ELSE
		standby := 15;
	END_IF
15:
		standbyCommand := TRUE;
		standby := 20;
20:
	standbyTimer(IN:= TRUE, PT := timeout);
	IF standbyTimer.Q THEN
		standbyTimer(IN:=FALSE);
		standby := 30;
	END_IF
30:

		IF standbyIncomplete OR NOT standbyStart THEN
			warningStandbyFailed := TRUE;
			standbyHalt := TRUE;
			IF  standbyClose THEN
				warningStandbyClose := TRUE;
			END_IF
		END_IF
		standby := 40;
40:

	standby := 900;

900:
	standby := 0;
END_CASE

(*-------------------------------------------------------------------------------------------------------------------------------------------*)

CASE third OF
0:
	IF startThird THEN
		third := 5;
	END_IF
5:
	IF thirdRemoteMode AND thirdAdditionalStat THEN
		third := 10;
	ELSE
		third := 900;
	END_IF
10:
	IF thirdOverload THEN
		warningThirdOverload := TRUE;
		thirdHalt := TRUE;
		third := 40;
	ELSE
		third := 15;
	END_IF
15:
		thirdCommand := TRUE;
		third := 20;
20:
	thirdTimer(IN:= TRUE, PT := timeout);
	IF thirdTimer.Q THEN
		thirdTimer(IN:=FALSE);
		third := 30;
	END_IF
30:

		IF thirdIncomplete OR NOT thirdStart THEN
			warningThirdFailed := TRUE;
			thirdHalt := TRUE;
			IF thirdClose THEN
				warningThirdClose := TRUE;
			END_IF
		END_IF
		third := 40;
40:

	third := 900;

900:
	third := 0;
END_CASE

(*-------------------------------------------------------------------------------------------------------------------------------------------*)

ROnce5(CLK:=(state=5));
IF ROnce5.Q THEN
		A1^:= TRUE;
		A2^:=TRUE;
		A3^ :=TRUE;
END_IF

ROnce10(CLK:=(state=10));
IF ROnce10.Q THEN
		B1^:= TRUE;
		B2^:= TRUE;
		B3^:= TRUE;
END_IF

IF thirdDevice THEN
ROnce20(CLK:=(state=20));
IF ROnce20.Q THEN
		C1^:= TRUE;
		C2^:= TRUE;
		C3^:= TRUE;
END_IF
END_IF

(*-------------------------------------------------------------------------------------------------------------------------------------------*)
GuardTONDuty(IN:=dutyIncomplete OR dutyOverload OR NOT dutyStart, PT:= GuardTime);
IF GuardTONDuty.Q THEN
	G1^ := TRUE;
END_IF
GuardTONStandby(IN:=standbyIncomplete OR standbyOverload OR NOT standbyStart, PT:= GuardTime);
IF GuardTONStandby.Q THEN
	G2^ := TRUE;
END_IF

IF thirdDevice THEN
GuardTONThird(IN:=thirdIncomplete OR thirdOverload OR NOT thirdStart, PT:= GuardTime);
IF GuardTONThird.q THEN
	G3^ := TRUE;
END_IF
END_IF
(*-------------------------------------------------------------------------------------------------------------------------------------------*)
stopAction;
test();
END_FUNCTION_BLOCK
ACTION stopAction:
CASE iStopDuty OF
0:
	DutyStopR(CLK:=stopDuty);
	IF DutyStopR.Q THEN
		iStopDuty := 5;
	END_IF
5:
	IF FSMode THEN
		FSStopDuty(IN:=TRUE,PT:=FSTime);
		IF FSStopDuty.Q THEN
			iStopDuty := 10;
			FSStopDuty(IN:=FALSE,PT:=FSTime);
		END_IF
	ELSE
		iStopDuty:=10;
	END_IF
10:
	dutyCommand := FALSE;
	stopDutyTimer(IN:=TRUE, PT:=timeout);
		IF stopDutyTimer.Q THEN
			stopDutyTimer(IN:=FALSE);
			IF NOT dutyClose THEN
				IF dutyStart THEN
					criticalDutyStopFailed := TRUE;
				END_IF
				warningDutyNotClose := TRUE;
			END_IF
			iStopDuty := 0;
		END_IF
END_CASE

(*-------------------------------------------------------------------------------------------------------------------------------------------*)

CASE iStopStandby OF
0:
	StandbyStopR(CLK:=stopStandby);
	IF StandbyStopR.Q THEN
		iStopStandby := 5;
	END_IF
5:
	IF FSMode THEN
		FSStopStandby(IN:=TRUE,PT:=FSTime);
		IF FSStopStandby.Q THEN
			iStopStandby := 10;
			FSStopStandby(IN:=FALSE,PT:=FSTime);
		END_IF
	ELSE
		iStopStandby:=10;
	END_IF
10:
	standbyCommand := FALSE;
	stopStandbyTimer(IN:=TRUE, PT:=timeout);
		IF stopStandbyTimer.Q THEN
			stopStandbyTimer(IN:=FALSE);
			IF NOT standbyClose THEN
				IF standbyStart THEN
					criticalStandbyStopFailed := TRUE;
				END_IF
					warningStandbyNotClose := TRUE;
			END_IF
			iStopStandby := 0;
		END_IF
END_CASE


(*-------------------------------------------------------------------------------------------------------------------------------------------*)

CASE iStopThird OF
0:
	ThirdStopR(CLK:=stopThird);
	IF ThirdStopR.Q THEN
		iStopThird := 10;
	END_IF
10:
	thirdCommand := FALSE;
	stopThirdTimer(IN:=TRUE, PT:=timeout);
		IF stopThirdTimer.Q THEN
			stopThirdTimer(IN:=FALSE);
			IF NOT thirdClose THEN
				IF thirdStart THEN
					criticalThirdStopFailed := TRUE;
				END_IF
				warningThirdNotClose := TRUE;
			END_IF
			iStopThird := 0;
		END_IF
END_CASE


(*-------------------------------------------------------------------------------------------------------------------------------------------*)

SOnceDuty(CLK:=(iStopDuty = 10));
IF SOnceDuty.Q THEN
		A1^:=FALSE;
		A2^:=FALSE;
		A3^:=FALSE;
END_IF


SOnceStandby(CLK:=(iStopStandby = 10));
IF SOnceStandby.Q THEN
		B1^:=FALSE;
		B2^:=FALSE;
		B3^:=FALSE;
END_IF

IF thirdDevice THEN
SOnceThird(CLK:=(iStopThird = 10));
IF SOnceThird.Q THEN
		C1^:=FALSE;
		C2^:=FALSE;
		C3^:=FALSE;
END_IF
END_IF


(*-------------------------------------------------------------------------------------------------------------------------------------------*)

(*
IF FSMode THEN

FSBothStop(IN:=NOT dutyCommand AND NOT standbyCommand,PT:=FSBothTime);
SOnceFS(CLK:=FSBothStop.Q);
IF SOnceFS.Q THEN
	FSBothStop(IN:=FALSE,PT:=FSBothTime);
	Q1^ := TRUE;
	Q2^ := TRUE;
	Q3^:=TRUE;
END_IF

END_IF
*)
END_ACTION
ACTION test:
dutyStart := dutyCommand;
standbyStart := standbyCommand;
thirdStart:=thirdCommand;
END_ACTION

(* POU module/trigBlock, ST *)
FUNCTION_BLOCK trigBlock
VAR_INPUT
	IN:BOOL;
	aQ:POINTER TO BOOL;
END_VAR
VAR_OUTPUT
END_VAR
VAR
	inR_TRIG: R_TRIG;
	outF_TRIG: F_TRIG;
	Q: BOOL;
END_VAR
VAR_IN_OUT
END_VAR
IF aQ = 0 THEN
	aQ := ADR(Q);
END_IF


inR_TRIG(CLK:=IN );
outF_TRIG(CLK:=IN );

IF inR_TRIG.Q THEN
	aQ^ := TRUE;
ELSIF  outF_TRIG.Q THEN
	aQ^ := FALSE;
END_IF
END_FUNCTION_BLOCK
